LIN {X -15.690,Y -24.253,Z -48.585,A -90.000,B 90.000,C 0.000} C_DIS
LIN {X -14.979,Y -24.271,Z -48.414,A -90.000,B 90.000,C 0.000} C_DIS
LIN {X -14.534,Y -24.273,Z -48.316,A -90.000,B 90.000,C 0.000} C_DIS
LIN {X -13.675,Y -24.281,Z -48.156,A -90.000,B 90.000,C 0.000} C_DIS
LIN {X -13.403,Y -24.283,Z -48.108,A -90.000,B 90.000,C 0.000} C_DIS
LIN {X -13.192,Y -24.287,Z -48.076,A -90.000,B 90.000,C 0.000} C_DIS
LIN {X -13.001,Y -24.291,Z -48.054,A -90.000,B 90.000,C 0.000} C_DIS
LIN {X -12.088,Y -24.285,Z -47.948,A -90.000,B 90.000,C 0.000} C_DIS
LIN {X -11.996,Y -24.284,Z -47.939,A -90.000,B 90.000,C 0.000} C_DIS
LIN {X -10.985,Y -24.286,Z -47.870,A -90.000,B 90.000,C 0.000} C_DIS
LIN {X -10.430,Y -24.283,Z -47.833,A -90.000,B 90.000,C 0.000} C_DIS
LIN {X -10.008,Y -24.276,Z -47.814,A -90.000,B 90.000,C 0.000} C_DIS
LIN {X -9.074,Y -24.265,Z -47.794,A -90.000,B 90.000,C 0.000} C_DIS
LIN {X -8.874,Y -24.263,Z -47.795,A -90.000,B 90.000,C 0.000} C_DIS
LIN {X -8.324,Y -24.259,Z -47.794,A -90.000,B 90.000,C 0.000} C_DIS
LIN {X -8.099,Y -24.253,Z -47.798,A -90.000,B 90.000,C 0.000} C_DIS
LIN {X -6.871,Y -24.218,Z -47.835,A -90.000,B 90.000,C 0.000} C_DIS
LIN {X -5.951,Y -24.176,Z -47.868,A -90.000,B 90.000,C 0.000} C_DIS
LIN {X -5.359,Y -24.150,Z -47.900,A -90.000,B 90.000,C 0.000} C_DIS
LIN {X -3.919,Y -24.078,Z -48.003,A -90.000,B 90.000,C 0.000} C_DIS
LIN {X -3.281,Y -24.035,Z -48.050,A -90.000,B 90.000,C 0.000} C_DIS
LIN {X -3.006,Y -24.019,Z -48.078,A -90.000,B 90.000,C 0.000} C_DIS
LIN {X -2.826,Y -24.007,Z -48.091,A -90.000,B 90.000,C 0.000} C_DIS
LIN {X -2.559,Y -23.983,Z -48.112,A -90.000,B 90.000,C 0.000} C_DIS
LIN {X -1.553,Y -23.901,Z -48.211,A -90.000,B 90.000,C 0.000} C_DIS
LIN {X -0.357,Y -23.796,Z -48.335,A -90.000,B 90.000,C 0.000} C_DIS
LIN {X -0.072,Y -23.770,Z -48.373,A -90.000,B 90.000,C 0.000} C_DIS
LIN {X 0.616,Y -23.686,Z -48.423,A -90.000,B 90.000,C 0.000} C_DIS
LIN {X 0.820,Y -23.658,Z -48.442,A -90.000,B 90.000,C 0.000} C_DIS
LIN {X 1.112,Y -23.624,Z -48.468,A -90.000,B 90.000,C 0.000} C_DIS
LIN {X 1.553,Y -23.560,Z -48.482,A -90.000,B 90.000,C 0.000} C_DIS
LIN {X 2.189,Y -23.460,Z -48.509,A -90.000,B 90.000,C 0.000} C_DIS
LIN {X 2.579,Y -23.392,Z -48.514,A -90.000,B 90.000,C 0.000} C_DIS
LIN {X 3.096,Y -23.308,Z -48.519,A -90.000,B 90.000,C 0.000} C_DIS
LIN {X 3.096,Y -60.000,Z -48.519,A -90.000,B 90.000,C 0.000} C_DIS
LIN {X -32.585,Y -60.000,Z -45.788,A -90.000,B 90.000,C 0.000} C_DIS
LIN {X -32.585,Y -23.308,Z -45.788,A -90.000,B 90.000,C 0.000} C_DIS
LIN {X -32.505,Y -23.313,Z -45.784,A -90.000,B 90.000,C 0.000} C_DIS
LIN {X -31.998,Y -23.345,Z -45.829,A -90.000,B 90.000,C 0.000} C_DIS
LIN {X -31.484,Y -23.377,Z -45.944,A -90.000,B 90.000,C 0.000} C_DIS
LIN {X -30.921,Y -23.413,Z -46.084,A -90.000,B 90.000,C 0.000} C_DIS
LIN {X -30.620,Y -23.432,Z -46.161,A -90.000,B 90.000,C 0.000} C_DIS
LIN {X -29.471,Y -23.490,Z -46.457,A -90.000,B 90.000,C 0.000} C_DIS
LIN {X -28.623,Y -23.534,Z -46.679,A -90.000,B 90.000,C 0.000} C_DIS
LIN {X -27.966,Y -23.569,Z -46.858,A -90.000,B 90.000,C 0.000} C_DIS
LIN {X -27.371,Y -23.600,Z -47.027,A -90.000,B 90.000,C 0.000} C_DIS
LIN {X -26.595,Y -23.630,Z -47.249,A -90.000,B 90.000,C 0.000} C_DIS
LIN {X -25.870,Y -23.674,Z -47.454,A -90.000,B 90.000,C 0.000} C_DIS
LIN {X -24.845,Y -23.735,Z -47.733,A -90.000,B 90.000,C 0.000} C_DIS
LIN {X -24.579,Y -23.747,Z -47.807,A -90.000,B 90.000,C 0.000} C_DIS
LIN {X -23.879,Y -23.794,Z -48.000,A -90.000,B 90.000,C 0.000} C_DIS
LIN {X -23.725,Y -23.804,Z -48.041,A -90.000,B 90.000,C 0.000} C_DIS
LIN {X -22.667,Y -23.874,Z -48.311,A -90.000,B 90.000,C 0.000} C_DIS
LIN {X -22.222,Y -23.905,Z -48.432,A -90.000,B 90.000,C 0.000} C_DIS
LIN {X -21.863,Y -23.929,Z -48.510,A -90.000,B 90.000,C 0.000} C_DIS
LIN {X -21.455,Y -23.955,Z -48.592,A -90.000,B 90.000,C 0.000} C_DIS
LIN {X -21.255,Y -23.968,Z -48.635,A -90.000,B 90.000,C 0.000} C_DIS
LIN {X -21.041,Y -23.972,Z -48.532,A -90.000,B 90.000,C 0.000} C_DIS
LIN {X -20.633,Y -23.979,Z -48.352,A -90.000,B 90.000,C 0.000} C_DIS
LIN {X -20.360,Y -23.979,Z -48.218,A -90.000,B 90.000,C 0.000} C_DIS
LIN {X -19.794,Y -23.981,Z -47.962,A -90.000,B 90.000,C 0.000} C_DIS
LIN {X -19.288,Y -23.984,Z -47.740,A -90.000,B 90.000,C 0.000} C_DIS
LIN {X -18.693,Y -23.989,Z -47.495,A -90.000,B 90.000,C 0.000} C_DIS
LIN {X -18.571,Y -23.990,Z -47.448,A -90.000,B 90.000,C 0.000} C_DIS
LIN {X -18.128,Y -23.997,Z -47.278,A -90.000,B 90.000,C 0.000} C_DIS
LIN {X -17.827,Y -23.998,Z -47.165,A -90.000,B 90.000,C 0.000} C_DIS
LIN {X -17.635,Y -23.992,Z -47.095,A -90.000,B 90.000,C 0.000} C_DIS
LIN {X -17.171,Y -23.976,Z -46.936,A -90.000,B 90.000,C 0.000} C_DIS
LIN {X -16.972,Y -23.970,Z -46.873,A -90.000,B 90.000,C 0.000} C_DIS
LIN {X -16.791,Y -23.966,Z -46.823,A -90.000,B 90.000,C 0.000} C_DIS
LIN {X -16.610,Y -23.962,Z -46.776,A -90.000,B 90.000,C 0.000} C_DIS
LIN {X -16.390,Y -23.958,Z -46.723,A -90.000,B 90.000,C 0.000} C_DIS
LIN {X -16.098,Y -23.953,Z -46.650,A -90.000,B 90.000,C 0.000} C_DIS
LIN {X -15.459,Y -23.940,Z -46.501,A -90.000,B 90.000,C 0.000} C_DIS
LIN {X -14.891,Y -23.930,Z -46.378,A -90.000,B 90.000,C 0.000} C_DIS
LIN {X -14.327,Y -23.923,Z -46.276,A -90.000,B 90.000,C 0.000} C_DIS
LIN {X -14.012,Y -23.915,Z -46.219,A -90.000,B 90.000,C 0.000} C_DIS
LIN {X -13.695,Y -23.908,Z -46.166,A -90.000,B 90.000,C 0.000} C_DIS
LIN {X -13.405,Y -23.902,Z -46.125,A -90.000,B 90.000,C 0.000} C_DIS
LIN {X -12.856,Y -23.894,Z -46.063,A -90.000,B 90.000,C 0.000} C_DIS
LIN {X -12.269,Y -23.874,Z -45.999,A -90.000,B 90.000,C 0.000} C_DIS
LIN {X -12.130,Y -23.869,Z -45.988,A -90.000,B 90.000,C 0.000} C_DIS
LIN {X -11.523,Y -23.849,Z -45.950,A -90.000,B 90.000,C 0.000} C_DIS
LIN {X -10.523,Y -23.813,Z -45.891,A -90.000,B 90.000,C 0.000} C_DIS
LIN {X -10.335,Y -23.807,Z -45.884,A -90.000,B 90.000,C 0.000} C_DIS
LIN {X -10.056,Y -23.794,Z -45.874,A -90.000,B 90.000,C 0.000} C_DIS
LIN {X -9.071,Y -23.756,Z -45.860,A -90.000,B 90.000,C 0.000} C_DIS
LIN {X -8.242,Y -23.727,Z -45.867,A -90.000,B 90.000,C 0.000} C_DIS
LIN {X -7.898,Y -23.712,Z -45.877,A -90.000,B 90.000,C 0.000} C_DIS
LIN {X -6.829,Y -23.656,Z -45.916,A -90.000,B 90.000,C 0.000} C_DIS
LIN {X -5.872,Y -23.593,Z -45.956,A -90.000,B 90.000,C 0.000} C_DIS
LIN {X -5.253,Y -23.547,Z -45.996,A -90.000,B 90.000,C 0.000} C_DIS
LIN {X -4.815,Y -23.517,Z -46.030,A -90.000,B 90.000,C 0.000} C_DIS
LIN {X -3.187,Y -23.355,Z -46.172,A -90.000,B 90.000,C 0.000} C_DIS
LIN {X -2.890,Y -23.324,Z -46.206,A -90.000,B 90.000,C 0.000} C_DIS
LIN {X -2.747,Y -23.308,Z -46.218,A -90.000,B 90.000,C 0.000} C_DIS
LIN {X -2.747,Y -60.000,Z -46.218,A -90.000,B 90.000,C 0.000} C_DIS
LIN {X -28.775,Y -60.000,Z -44.581,A -90.000,B 90.000,C 0.000} C_DIS
LIN {X -28.775,Y -23.308,Z -44.581,A -90.000,B 90.000,C 0.000} C_DIS
LIN {X -27.940,Y -23.354,Z -44.801,A -90.000,B 90.000,C 0.000} C_DIS
LIN {X -27.677,Y -23.366,Z -44.873,A -90.000,B 90.000,C 0.000} C_DIS
LIN {X -27.412,Y -23.377,Z -44.946,A -90.000,B 90.000,C 0.000} C_DIS
LIN {X -26.438,Y -23.416,Z -45.224,A -90.000,B 90.000,C 0.000} C_DIS
LIN {X -25.243,Y -23.500,Z -45.560,A -90.000,B 90.000,C 0.000} C_DIS
LIN {X -24.377,Y -23.540,Z -45.797,A -90.000,B 90.000,C 0.000} C_DIS
LIN {X -23.210,Y -23.631,Z -46.116,A -90.000,B 90.000,C 0.000} C_DIS
LIN {X -22.965,Y -23.648,Z -46.179,A -90.000,B 90.000,C 0.000} C_DIS
LIN {X -22.513,Y -23.673,Z -46.294,A -90.000,B 90.000,C 0.000} C_DIS
LIN {X -22.132,Y -23.703,Z -46.391,A -90.000,B 90.000,C 0.000} C_DIS
LIN {X -21.755,Y -23.733,Z -46.495,A -90.000,B 90.000,C 0.000} C_DIS
LIN {X -21.480,Y -23.754,Z -46.554,A -90.000,B 90.000,C 0.000} C_DIS
LIN {X -21.262,Y -23.752,Z -46.447,A -90.000,B 90.000,C 0.000} C_DIS
LIN {X -21.012,Y -23.750,Z -46.332,A -90.000,B 90.000,C 0.000} C_DIS
LIN {X -20.884,Y -23.746,Z -46.275,A -90.000,B 90.000,C 0.000} C_DIS
LIN {X -20.466,Y -23.723,Z -46.091,A -90.000,B 90.000,C 0.000} C_DIS
LIN {X -20.040,Y -23.701,Z -45.909,A -90.000,B 90.000,C 0.000} C_DIS
LIN {X -19.444,Y -23.672,Z -45.669,A -90.000,B 90.000,C 0.000} C_DIS
LIN {X -18.658,Y -23.639,Z -45.376,A -90.000,B 90.000,C 0.000} C_DIS
LIN {X -18.327,Y -23.625,Z -45.254,A -90.000,B 90.000,C 0.000} C_DIS
LIN {X -17.772,Y -23.605,Z -45.064,A -90.000,B 90.000,C 0.000} C_DIS
LIN {X -17.669,Y -23.602,Z -45.032,A -90.000,B 90.000,C 0.000} C_DIS
LIN {X -17.499,Y -23.597,Z -44.980,A -90.000,B 90.000,C 0.000} C_DIS
LIN {X -17.320,Y -23.592,Z -44.931,A -90.000,B 90.000,C 0.000} C_DIS
LIN {X -16.958,Y -23.568,Z -44.842,A -90.000,B 90.000,C 0.000} C_DIS
LIN {X -16.506,Y -23.540,Z -44.735,A -90.000,B 90.000,C 0.000} C_DIS
LIN {X -15.878,Y -23.503,Z -44.595,A -90.000,B 90.000,C 0.000} C_DIS
LIN {X -15.310,Y -23.472,Z -44.477,A -90.000,B 90.000,C 0.000} C_DIS
LIN {X -14.339,Y -23.429,Z -44.307,A -90.000,B 90.000,C 0.000} C_DIS
LIN {X -13.945,Y -23.412,Z -44.244,A -90.000,B 90.000,C 0.000} C_DIS
LIN {X -13.628,Y -23.395,Z -44.203,A -90.000,B 90.000,C 0.000} C_DIS
LIN {X -12.619,Y -23.342,Z -44.099,A -90.000,B 90.000,C 0.000} C_DIS
LIN {X -12.445,Y -23.328,Z -44.083,A -90.000,B 90.000,C 0.000} C_DIS
LIN {X -12.266,Y -23.316,Z -44.070,A -90.000,B 90.000,C 0.000} C_DIS
LIN {X -12.141,Y -23.308,Z -44.064,A -90.000,B 90.000,C 0.000} C_DIS
LIN {X -12.141,Y -60.000,Z -44.064,A -90.000,B 90.000,C 0.000} C_DIS
LIN {X -22.320,Y -60.000,Z -44.311,A -90.000,B 90.000,C 0.000} C_DIS
LIN {X -22.320,Y -23.308,Z -44.311,A -90.000,B 90.000,C 0.000} C_DIS
LIN {X -22.204,Y -23.316,Z -44.340,A -90.000,B 90.000,C 0.000} C_DIS
LIN {X -21.668,Y -23.364,Z -44.475,A -90.000,B 90.000,C 0.000} C_DIS
LIN {X -21.152,Y -23.332,Z -44.250,A -90.000,B 90.000,C 0.000} C_DIS
LIN {X -20.759,Y -23.308,Z -44.084,A -90.000,B 90.000,C 0.000} C_DIS
LIN {X -20.759,Y -60.000,Z -44.084,A -90.000,B 90.000,C 0.000} C_DIS
LIN {X -95.711,Y -60.000,Z -40.754,A -90.000,B 90.000,C 0.000} C_DIS
LIN {X -95.711,Y -23.308,Z -40.754,A -90.000,B 90.000,C 0.000} C_DIS
LIN {X -95.404,Y -23.376,Z -40.730,A -90.000,B 90.000,C 0.000} C_DIS
LIN {X -95.125,Y -23.439,Z -40.718,A -90.000,B 90.000,C 0.000} C_DIS
LIN {X -94.697,Y -23.539,Z -40.707,A -90.000,B 90.000,C 0.000} C_DIS
LIN {X -94.412,Y -23.607,Z -40.709,A -90.000,B 90.000,C 0.000} C_DIS
LIN {X -94.097,Y -23.689,Z -40.720,A -90.000,B 90.000,C 0.000} C_DIS
LIN {X -93.821,Y -23.753,Z -40.682,A -90.000,B 90.000,C 0.000} C_DIS
LIN {X -93.679,Y -23.787,Z -40.667,A -90.000,B 90.000,C 0.000} C_DIS
LIN {X -93.582,Y -23.810,Z -40.659,A -90.000,B 90.000,C 0.000} C_DIS
LIN {X -93.062,Y -23.940,Z -40.640,A -90.000,B 90.000,C 0.000} C_DIS
LIN {X -92.947,Y -23.969,Z -40.636,A -90.000,B 90.000,C 0.000} C_DIS
LIN {X -92.686,Y -24.037,Z -40.636,A -90.000,B 90.000,C 0.000} C_DIS
LIN {X -92.525,Y -24.079,Z -40.642,A -90.000,B 90.000,C 0.000} C_DIS
LIN {X -92.268,Y -24.147,Z -40.654,A -90.000,B 90.000,C 0.000} C_DIS
LIN {X -91.922,Y -24.239,Z -40.676,A -90.000,B 90.000,C 0.000} C_DIS
LIN {X -91.828,Y -24.217,Z -40.402,A -90.000,B 90.000,C 0.000} C_DIS
LIN {X -91.794,Y -24.207,Z -40.309,A -90.000,B 90.000,C 0.000} C_DIS
LIN {X -91.725,Y -24.191,Z -40.113,A -90.000,B 90.000,C 0.000} C_DIS
LIN {X -91.669,Y -24.181,Z -39.970,A -90.000,B 90.000,C 0.000} C_DIS
LIN {X -91.619,Y -24.175,Z -39.854,A -90.000,B 90.000,C 0.000} C_DIS
LIN {X -91.566,Y -24.169,Z -39.741,A -90.000,B 90.000,C 0.000} C_DIS
LIN {X -91.504,Y -24.165,Z -39.621,A -90.000,B 90.000,C 0.000} C_DIS
LIN {X -91.441,Y -24.153,Z -39.505,A -90.000,B 90.000,C 0.000} C_DIS
LIN {X -91.356,Y -24.139,Z -39.362,A -90.000,B 90.000,C 0.000} C_DIS
LIN {X -91.326,Y -24.131,Z -39.314,A -90.000,B 90.000,C 0.000} C_DIS
LIN {X -91.245,Y -24.118,Z -39.180,A -90.000,B 90.000,C 0.000} C_DIS
LIN {X -91.203,Y -24.112,Z -39.116,A -90.000,B 90.000,C 0.000} C_DIS
LIN {X -91.034,Y -24.087,Z -38.886,A -90.000,B 90.000,C 0.000} C_DIS
LIN {X -90.958,Y -24.072,Z -38.743,A -90.000,B 90.000,C 0.000} C_DIS
LIN {X -90.838,Y -24.039,Z -38.550,A -90.000,B 90.000,C 0.000} C_DIS
LIN {X -90.746,Y -24.015,Z -38.415,A -90.000,B 90.000,C 0.000} C_DIS
LIN {X -90.547,Y -23.961,Z -38.143,A -90.000,B 90.000,C 0.000} C_DIS
LIN {X -90.460,Y -23.947,Z -38.029,A -90.000,B 90.000,C 0.000} C_DIS
LIN {X -90.374,Y -23.936,Z -37.924,A -90.000,B 90.000,C 0.000} C_DIS
LIN {X -90.278,Y -23.926,Z -37.813,A -90.000,B 90.000,C 0.000} C_DIS
LIN {X -90.089,Y -23.895,Z -37.621,A -90.000,B 90.000,C 0.000} C_DIS
LIN {X -89.954,Y -23.869,Z -37.492,A -90.000,B 90.000,C 0.000} C_DIS
LIN {X -89.904,Y -23.863,Z -37.443,A -90.000,B 90.000,C 0.000} C_DIS
LIN {X -89.803,Y -23.853,Z -37.352,A -90.000,B 90.000,C 0.000} C_DIS
LIN {X -89.654,Y -23.839,Z -37.224,A -90.000,B 90.000,C 0.000} C_DIS
LIN {X -89.505,Y -23.828,Z -37.109,A -90.000,B 90.000,C 0.000} C_DIS
LIN {X -89.400,Y -23.817,Z -37.035,A -90.000,B 90.000,C 0.000} C_DIS
LIN {X -89.138,Y -23.799,Z -36.847,A -90.000,B 90.000,C 0.000} C_DIS
LIN {X -89.084,Y -23.790,Z -36.797,A -90.000,B 90.000,C 0.000} C_DIS
LIN {X -88.968,Y -23.771,Z -36.698,A -90.000,B 90.000,C 0.000} C_DIS
LIN {X -88.747,Y -23.744,Z -36.523,A -90.000,B 90.000,C 0.000} C_DIS
LIN {X -88.371,Y -23.709,Z -36.261,A -90.000,B 90.000,C 0.000} C_DIS
LIN {X -88.226,Y -23.699,Z -36.167,A -90.000,B 90.000,C 0.000} C_DIS
LIN {X -88.132,Y -23.696,Z -36.112,A -90.000,B 90.000,C 0.000} C_DIS
LIN {X -87.910,Y -23.694,Z -35.987,A -90.000,B 90.000,C 0.000} C_DIS
LIN {X -87.694,Y -23.697,Z -35.875,A -90.000,B 90.000,C 0.000} C_DIS
LIN {X -87.253,Y -23.682,Z -35.604,A -90.000,B 90.000,C 0.000} C_DIS
LIN {X -87.176,Y -23.680,Z -35.559,A -90.000,B 90.000,C 0.000} C_DIS
LIN {X -86.953,Y -23.677,Z -35.437,A -90.000,B 90.000,C 0.000} C_DIS
LIN {X -86.816,Y -23.677,Z -35.368,A -90.000,B 90.000,C 0.000} C_DIS
LIN {X -86.698,Y -23.684,Z -35.304,A -90.000,B 90.000,C 0.000} C_DIS
LIN {X -86.576,Y -23.704,Z -35.237,A -90.000,B 90.000,C 0.000} C_DIS
LIN {X -86.405,Y -23.727,Z -35.152,A -90.000,B 90.000,C 0.000} C_DIS
LIN {X -86.301,Y -23.742,Z -35.107,A -90.000,B 90.000,C 0.000} C_DIS
LIN {X -86.104,Y -23.770,Z -35.028,A -90.000,B 90.000,C 0.000} C_DIS
LIN {X -85.996,Y -23.785,Z -34.990,A -90.000,B 90.000,C 0.000} C_DIS
LIN {X -85.717,Y -23.820,Z -34.894,A -90.000,B 90.000,C 0.000} C_DIS
LIN {X -85.064,Y -23.902,Z -34.688,A -90.000,B 90.000,C 0.000} C_DIS
LIN {X -84.998,Y -23.910,Z -34.665,A -90.000,B 90.000,C 0.000} C_DIS
LIN {X -84.512,Y -23.958,Z -34.499,A -90.000,B 90.000,C 0.000} C_DIS
LIN {X -84.366,Y -23.973,Z -34.452,A -90.000,B 90.000,C 0.000} C_DIS
LIN {X -84.135,Y -23.992,Z -34.378,A -90.000,B 90.000,C 0.000} C_DIS
LIN {X -84.049,Y -24.002,Z -34.353,A -90.000,B 90.000,C 0.000} C_DIS
LIN {X -83.904,Y -24.017,Z -34.314,A -90.000,B 90.000,C 0.000} C_DIS
LIN {X -83.669,Y -24.044,Z -34.261,A -90.000,B 90.000,C 0.000} C_DIS
LIN {X -83.463,Y -24.068,Z -34.227,A -90.000,B 90.000,C 0.000} C_DIS
LIN {X -83.165,Y -24.104,Z -34.187,A -90.000,B 90.000,C 0.000} C_DIS
LIN {X -83.013,Y -24.122,Z -34.173,A -90.000,B 90.000,C 0.000} C_DIS
LIN {X -82.811,Y -24.142,Z -34.160,A -90.000,B 90.000,C 0.000} C_DIS
LIN {X -81.766,Y -24.254,Z -34.100,A -90.000,B 90.000,C 0.000} C_DIS
LIN {X -81.587,Y -24.268,Z -34.092,A -90.000,B 90.000,C 0.000} C_DIS
LIN {X -81.311,Y -24.285,Z -34.078,A -90.000,B 90.000,C 0.000} C_DIS
LIN {X -81.094,Y -24.301,Z -34.074,A -90.000,B 90.000,C 0.000} C_DIS
LIN {X -80.876,Y -24.317,Z -34.077,A -90.000,B 90.000,C 0.000} C_DIS
LIN {X -80.753,Y -24.325,Z -34.081,A -90.000,B 90.000,C 0.000} C_DIS
LIN {X -80.316,Y -24.356,Z -34.112,A -90.000,B 90.000,C 0.000} C_DIS
LIN {X -80.028,Y -24.375,Z -34.145,A -90.000,B 90.000,C 0.000} C_DIS
LIN {X -79.790,Y -24.379,Z -34.178,A -90.000,B 90.000,C 0.000} C_DIS
LIN {X -79.303,Y -24.376,Z -34.251,A -90.000,B 90.000,C 0.000} C_DIS
LIN {X -78.837,Y -24.372,Z -34.323,A -90.000,B 90.000,C 0.000} C_DIS
LIN {X -78.575,Y -24.369,Z -34.362,A -90.000,B 90.000,C 0.000} C_DIS
LIN {X -78.371,Y -24.366,Z -34.396,A -90.000,B 90.000,C 0.000} C_DIS
LIN {X -78.171,Y -24.360,Z -34.436,A -90.000,B 90.000,C 0.000} C_DIS
LIN {X -77.664,Y -24.319,Z -34.565,A -90.000,B 90.000,C 0.000} C_DIS
LIN {X -77.527,Y -24.308,Z -34.603,A -90.000,B 90.000,C 0.000} C_DIS
LIN {X -76.621,Y -24.210,Z -34.862,A -90.000,B 90.000,C 0.000} C_DIS
LIN {X -76.352,Y -24.182,Z -34.940,A -90.000,B 90.000,C 0.000} C_DIS
LIN {X -76.038,Y -24.153,Z -35.031,A -90.000,B 90.000,C 0.000} C_DIS
LIN {X -75.954,Y -24.146,Z -35.059,A -90.000,B 90.000,C 0.000} C_DIS
LIN {X -75.336,Y -24.059,Z -35.270,A -90.000,B 90.000,C 0.000} C_DIS
LIN {X -75.055,Y -24.015,Z -35.369,A -90.000,B 90.000,C 0.000} C_DIS
LIN {X -74.477,Y -23.967,Z -35.562,A -90.000,B 90.000,C 0.000} C_DIS
LIN {X -73.802,Y -23.909,Z -35.764,A -90.000,B 90.000,C 0.000} C_DIS
LIN {X -73.585,Y -23.884,Z -35.832,A -90.000,B 90.000,C 0.000} C_DIS
LIN {X -72.583,Y -23.813,Z -36.131,A -90.000,B 90.000,C 0.000} C_DIS
LIN {X -72.099,Y -23.794,Z -36.270,A -90.000,B 90.000,C 0.000} C_DIS
LIN {X -71.852,Y -23.780,Z -36.342,A -90.000,B 90.000,C 0.000} C_DIS
LIN {X -71.586,Y -23.758,Z -36.423,A -90.000,B 90.000,C 0.000} C_DIS
LIN {X -71.224,Y -23.733,Z -36.546,A -90.000,B 90.000,C 0.000} C_DIS
LIN {X -69.912,Y -23.680,Z -36.977,A -90.000,B 90.000,C 0.000} C_DIS
LIN {X -69.703,Y -23.674,Z -37.053,A -90.000,B 90.000,C 0.000} C_DIS
LIN {X -67.916,Y -23.609,Z -37.754,A -90.000,B 90.000,C 0.000} C_DIS
LIN {X -67.475,Y -23.601,Z -37.944,A -90.000,B 90.000,C 0.000} C_DIS
LIN {X -67.275,Y -23.600,Z -38.034,A -90.000,B 90.000,C 0.000} C_DIS
LIN {X -66.096,Y -23.581,Z -38.568,A -90.000,B 90.000,C 0.000} C_DIS
LIN {X -65.374,Y -23.570,Z -38.895,A -90.000,B 90.000,C 0.000} C_DIS
LIN {X -65.123,Y -23.567,Z -39.012,A -90.000,B 90.000,C 0.000} C_DIS
LIN {X -64.632,Y -23.569,Z -39.237,A -90.000,B 90.000,C 0.000} C_DIS
LIN {X -63.049,Y -23.568,Z -39.976,A -90.000,B 90.000,C 0.000} C_DIS
LIN {X -62.587,Y -23.563,Z -40.182,A -90.000,B 90.000,C 0.000} C_DIS
LIN {X -61.622,Y -23.570,Z -40.601,A -90.000,B 90.000,C 0.000} C_DIS
LIN {X -60.883,Y -23.573,Z -40.925,A -90.000,B 90.000,C 0.000} C_DIS
LIN {X -59.965,Y -23.555,Z -41.283,A -90.000,B 90.000,C 0.000} C_DIS
LIN {X -58.440,Y -23.556,Z -41.863,A -90.000,B 90.000,C 0.000} C_DIS
LIN {X -57.686,Y -23.533,Z -42.100,A -90.000,B 90.000,C 0.000} C_DIS
LIN {X -57.271,Y -23.524,Z -42.228,A -90.000,B 90.000,C 0.000} C_DIS
LIN {X -56.299,Y -23.512,Z -42.523,A -90.000,B 90.000,C 0.000} C_DIS
LIN {X -55.979,Y -23.509,Z -42.624,A -90.000,B 90.000,C 0.000} C_DIS
LIN {X -54.824,Y -23.462,Z -42.911,A -90.000,B 90.000,C 0.000} C_DIS
LIN {X -54.566,Y -23.454,Z -42.978,A -90.000,B 90.000,C 0.000} C_DIS
LIN {X -53.632,Y -23.437,Z -43.217,A -90.000,B 90.000,C 0.000} C_DIS
LIN {X -53.189,Y -23.414,Z -43.304,A -90.000,B 90.000,C 0.000} C_DIS
LIN {X -52.188,Y -23.372,Z -43.522,A -90.000,B 90.000,C 0.000} C_DIS
LIN {X -51.677,Y -23.361,Z -43.648,A -90.000,B 90.000,C 0.000} C_DIS
LIN {X -50.718,Y -23.347,Z -43.882,A -90.000,B 90.000,C 0.000} C_DIS
LIN {X -50.007,Y -23.330,Z -44.041,A -90.000,B 90.000,C 0.000} C_DIS
LIN {X -49.018,Y -23.308,Z -44.257,A -90.000,B 90.000,C 0.000} C_DIS
LIN {X -49.018,Y -60.000,Z -44.257,A -90.000,B 90.000,C 0.000} C_DIS
LIN {X -88.889,Y -60.000,Z -34.286,A -90.000,B 90.000,C 0.000} C_DIS
LIN {X -88.889,Y -23.308,Z -34.286,A -90.000,B 90.000,C 0.000} C_DIS
LIN {X -88.778,Y -23.327,Z -34.222,A -90.000,B 90.000,C 0.000} C_DIS
LIN {X -88.666,Y -23.346,Z -34.161,A -90.000,B 90.000,C 0.000} C_DIS
LIN {X -88.534,Y -23.367,Z -34.075,A -90.000,B 90.000,C 0.000} C_DIS
LIN {X -88.241,Y -23.405,Z -33.888,A -90.000,B 90.000,C 0.000} C_DIS
LIN {X -88.132,Y -23.419,Z -33.822,A -90.000,B 90.000,C 0.000} C_DIS
LIN {X -87.851,Y -23.453,Z -33.664,A -90.000,B 90.000,C 0.000} C_DIS
LIN {X -87.674,Y -23.475,Z -33.571,A -90.000,B 90.000,C 0.000} C_DIS
LIN {X -87.558,Y -23.485,Z -33.508,A -90.000,B 90.000,C 0.000} C_DIS
LIN {X -87.382,Y -23.494,Z -33.417,A -90.000,B 90.000,C 0.000} C_DIS
LIN {X -87.268,Y -23.500,Z -33.362,A -90.000,B 90.000,C 0.000} C_DIS
LIN {X -87.116,Y -23.508,Z -33.294,A -90.000,B 90.000,C 0.000} C_DIS
LIN {X -86.979,Y -23.516,Z -33.238,A -90.000,B 90.000,C 0.000} C_DIS
LIN {X -86.761,Y -23.529,Z -33.155,A -90.000,B 90.000,C 0.000} C_DIS
LIN {X -86.511,Y -23.545,Z -33.069,A -90.000,B 90.000,C 0.000} C_DIS
LIN {X -86.235,Y -23.568,Z -32.978,A -90.000,B 90.000,C 0.000} C_DIS
LIN {X -85.622,Y -23.609,Z -32.788,A -90.000,B 90.000,C 0.000} C_DIS
LIN {X -85.221,Y -23.633,Z -32.655,A -90.000,B 90.000,C 0.000} C_DIS
LIN {X -84.885,Y -23.675,Z -32.542,A -90.000,B 90.000,C 0.000} C_DIS
LIN {X -84.715,Y -23.696,Z -32.487,A -90.000,B 90.000,C 0.000} C_DIS
LIN {X -84.589,Y -23.712,Z -32.449,A -90.000,B 90.000,C 0.000} C_DIS
LIN {X -84.319,Y -23.747,Z -32.376,A -90.000,B 90.000,C 0.000} C_DIS
LIN {X -84.073,Y -23.788,Z -32.319,A -90.000,B 90.000,C 0.000} C_DIS
LIN {X -83.965,Y -23.806,Z -32.298,A -90.000,B 90.000,C 0.000} C_DIS
LIN {X -83.702,Y -23.850,Z -32.253,A -90.000,B 90.000,C 0.000} C_DIS
LIN {X -83.406,Y -23.900,Z -32.212,A -90.000,B 90.000,C 0.000} C_DIS
LIN {X -83.176,Y -23.940,Z -32.188,A -90.000,B 90.000,C 0.000} C_DIS
LIN {X -82.798,Y -24.007,Z -32.161,A -90.000,B 90.000,C 0.000} C_DIS
LIN {X -82.322,Y -24.090,Z -32.132,A -90.000,B 90.000,C 0.000} C_DIS
LIN {X -81.879,Y -24.162,Z -32.105,A -90.000,B 90.000,C 0.000} C_DIS
LIN {X -81.618,Y -24.203,Z -32.092,A -90.000,B 90.000,C 0.000} C_DIS
LIN {X -81.411,Y -24.229,Z -32.082,A -90.000,B 90.000,C 0.000} C_DIS
LIN {X -81.065,Y -24.268,Z -32.074,A -90.000,B 90.000,C 0.000} C_DIS
LIN {X -80.767,Y -24.303,Z -32.079,A -90.000,B 90.000,C 0.000} C_DIS
LIN {X -80.612,Y -24.323,Z -32.086,A -90.000,B 90.000,C 0.000} C_DIS
LIN {X -80.222,Y -24.371,Z -32.114,A -90.000,B 90.000,C 0.000} C_DIS
LIN {X -80.090,Y -24.383,Z -32.125,A -90.000,B 90.000,C 0.000} C_DIS
LIN {X -79.758,Y -24.412,Z -32.164,A -90.000,B 90.000,C 0.000} C_DIS
LIN {X -79.546,Y -24.429,Z -32.193,A -90.000,B 90.000,C 0.000} C_DIS
LIN {X -79.200,Y -24.444,Z -32.245,A -90.000,B 90.000,C 0.000} C_DIS
LIN {X -79.004,Y -24.448,Z -32.275,A -90.000,B 90.000,C 0.000} C_DIS
LIN {X -78.188,Y -24.442,Z -32.400,A -90.000,B 90.000,C 0.000} C_DIS
LIN {X -78.032,Y -24.438,Z -32.426,A -90.000,B 90.000,C 0.000} C_DIS
LIN {X -77.969,Y -24.434,Z -32.438,A -90.000,B 90.000,C 0.000} C_DIS
LIN {X -77.785,Y -24.419,Z -32.474,A -90.000,B 90.000,C 0.000} C_DIS
LIN {X -77.638,Y -24.407,Z -32.508,A -90.000,B 90.000,C 0.000} C_DIS
LIN {X -77.098,Y -24.355,Z -32.647,A -90.000,B 90.000,C 0.000} C_DIS
LIN {X -76.573,Y -24.302,Z -32.796,A -90.000,B 90.000,C 0.000} C_DIS
LIN {X -76.436,Y -24.283,Z -32.835,A -90.000,B 90.000,C 0.000} C_DIS
LIN {X -76.069,Y -24.222,Z -32.940,A -90.000,B 90.000,C 0.000} C_DIS
LIN {X -75.819,Y -24.176,Z -33.012,A -90.000,B 90.000,C 0.000} C_DIS
LIN {X -75.618,Y -24.137,Z -33.071,A -90.000,B 90.000,C 0.000} C_DIS
LIN {X -75.424,Y -24.099,Z -33.129,A -90.000,B 90.000,C 0.000} C_DIS
LIN {X -75.182,Y -24.043,Z -33.211,A -90.000,B 90.000,C 0.000} C_DIS
LIN {X -74.616,Y -23.897,Z -33.409,A -90.000,B 90.000,C 0.000} C_DIS
LIN {X -73.871,Y -23.698,Z -33.674,A -90.000,B 90.000,C 0.000} C_DIS
LIN {X -73.225,Y -23.527,Z -33.888,A -90.000,B 90.000,C 0.000} C_DIS
LIN {X -73.049,Y -23.476,Z -33.949,A -90.000,B 90.000,C 0.000} C_DIS
LIN {X -72.827,Y -23.429,Z -34.022,A -90.000,B 90.000,C 0.000} C_DIS
LIN {X -72.333,Y -23.308,Z -34.192,A -90.000,B 90.000,C 0.000} C_DIS
LIN {X -72.333,Y -60.000,Z -34.192,A -90.000,B 90.000,C 0.000} C_DIS
LIN {X -85.759,Y -60.000,Z -30.755,A -90.000,B 90.000,C 0.000} C_DIS
LIN {X -85.759,Y -23.308,Z -30.755,A -90.000,B 90.000,C 0.000} C_DIS
LIN {X -85.664,Y -23.324,Z -30.723,A -90.000,B 90.000,C 0.000} C_DIS
LIN {X -85.255,Y -23.408,Z -30.583,A -90.000,B 90.000,C 0.000} C_DIS
LIN {X -85.054,Y -23.450,Z -30.521,A -90.000,B 90.000,C 0.000} C_DIS
LIN {X -84.801,Y -23.506,Z -30.450,A -90.000,B 90.000,C 0.000} C_DIS
LIN {X -84.485,Y -23.575,Z -30.374,A -90.000,B 90.000,C 0.000} C_DIS
LIN {X -84.265,Y -23.623,Z -30.329,A -90.000,B 90.000,C 0.000} C_DIS
LIN {X -83.951,Y -23.691,Z -30.275,A -90.000,B 90.000,C 0.000} C_DIS
LIN {X -83.592,Y -23.772,Z -30.225,A -90.000,B 90.000,C 0.000} C_DIS
LIN {X -83.381,Y -23.815,Z -30.202,A -90.000,B 90.000,C 0.000} C_DIS
LIN {X -82.958,Y -23.893,Z -30.171,A -90.000,B 90.000,C 0.000} C_DIS
LIN {X -81.890,Y -24.094,Z -30.105,A -90.000,B 90.000,C 0.000} C_DIS
LIN {X -81.695,Y -24.131,Z -30.095,A -90.000,B 90.000,C 0.000} C_DIS
LIN {X -81.520,Y -24.159,Z -30.086,A -90.000,B 90.000,C 0.000} C_DIS
LIN {X -81.082,Y -24.218,Z -30.075,A -90.000,B 90.000,C 0.000} C_DIS
LIN {X -80.676,Y -24.270,Z -30.082,A -90.000,B 90.000,C 0.000} C_DIS
LIN {X -80.467,Y -24.296,Z -30.092,A -90.000,B 90.000,C 0.000} C_DIS
LIN {X -80.079,Y -24.339,Z -30.119,A -90.000,B 90.000,C 0.000} C_DIS
LIN {X -79.860,Y -24.360,Z -30.138,A -90.000,B 90.000,C 0.000} C_DIS
LIN {X -79.410,Y -24.393,Z -30.193,A -90.000,B 90.000,C 0.000} C_DIS
LIN {X -78.795,Y -24.430,Z -30.284,A -90.000,B 90.000,C 0.000} C_DIS
LIN {X -78.735,Y -24.434,Z -30.293,A -90.000,B 90.000,C 0.000} C_DIS
LIN {X -78.394,Y -24.455,Z -30.345,A -90.000,B 90.000,C 0.000} C_DIS
LIN {X -78.090,Y -24.460,Z -30.392,A -90.000,B 90.000,C 0.000} C_DIS
LIN {X -77.830,Y -24.457,Z -30.432,A -90.000,B 90.000,C 0.000} C_DIS
LIN {X -77.584,Y -24.445,Z -30.475,A -90.000,B 90.000,C 0.000} C_DIS
LIN {X -77.332,Y -24.434,Z -30.526,A -90.000,B 90.000,C 0.000} C_DIS
LIN {X -77.140,Y -24.425,Z -30.571,A -90.000,B 90.000,C 0.000} C_DIS
LIN {X -76.598,Y -24.385,Z -30.710,A -90.000,B 90.000,C 0.000} C_DIS
LIN {X -76.167,Y -24.349,Z -30.832,A -90.000,B 90.000,C 0.000} C_DIS
LIN {X -75.917,Y -24.323,Z -30.904,A -90.000,B 90.000,C 0.000} C_DIS
LIN {X -75.829,Y -24.311,Z -30.929,A -90.000,B 90.000,C 0.000} C_DIS
LIN {X -75.368,Y -24.220,Z -31.061,A -90.000,B 90.000,C 0.000} C_DIS
LIN {X -75.188,Y -24.179,Z -31.113,A -90.000,B 90.000,C 0.000} C_DIS
LIN {X -74.888,Y -24.098,Z -31.202,A -90.000,B 90.000,C 0.000} C_DIS
LIN {X -74.796,Y -24.072,Z -31.230,A -90.000,B 90.000,C 0.000} C_DIS
LIN {X -74.517,Y -23.994,Z -31.325,A -90.000,B 90.000,C 0.000} C_DIS
LIN {X -74.060,Y -23.866,Z -31.486,A -90.000,B 90.000,C 0.000} C_DIS
LIN {X -73.848,Y -23.801,Z -31.561,A -90.000,B 90.000,C 0.000} C_DIS
LIN {X -73.462,Y -23.679,Z -31.699,A -90.000,B 90.000,C 0.000} C_DIS
LIN {X -73.247,Y -23.603,Z -31.776,A -90.000,B 90.000,C 0.000} C_DIS
LIN {X -72.844,Y -23.462,Z -31.911,A -90.000,B 90.000,C 0.000} C_DIS
LIN {X -72.608,Y -23.375,Z -31.991,A -90.000,B 90.000,C 0.000} C_DIS
LIN {X -72.432,Y -23.308,Z -32.054,A -90.000,B 90.000,C 0.000} C_DIS
LIN {X -72.432,Y -60.000,Z -32.054,A -90.000,B 90.000,C 0.000} C_DIS
LIN {X -86.147,Y -60.000,Z -28.775,A -90.000,B 90.000,C 0.000} C_DIS
LIN {X -86.147,Y -23.308,Z -28.775,A -90.000,B 90.000,C 0.000} C_DIS
LIN {X -85.995,Y -23.351,Z -28.723,A -90.000,B 90.000,C 0.000} C_DIS
LIN {X -85.792,Y -23.399,Z -28.656,A -90.000,B 90.000,C 0.000} C_DIS
LIN {X -85.596,Y -23.444,Z -28.596,A -90.000,B 90.000,C 0.000} C_DIS
LIN {X -85.272,Y -23.518,Z -28.506,A -90.000,B 90.000,C 0.000} C_DIS
LIN {X -85.011,Y -23.577,Z -28.443,A -90.000,B 90.000,C 0.000} C_DIS
LIN {X -84.891,Y -23.600,Z -28.416,A -90.000,B 90.000,C 0.000} C_DIS
LIN {X -84.606,Y -23.654,Z -28.358,A -90.000,B 90.000,C 0.000} C_DIS
LIN {X -84.235,Y -23.723,Z -28.296,A -90.000,B 90.000,C 0.000} C_DIS
LIN {X -83.810,Y -23.800,Z -28.237,A -90.000,B 90.000,C 0.000} C_DIS
LIN {X -83.535,Y -23.844,Z -28.209,A -90.000,B 90.000,C 0.000} C_DIS
LIN {X -83.437,Y -23.859,Z -28.201,A -90.000,B 90.000,C 0.000} C_DIS
LIN {X -83.081,Y -23.895,Z -28.175,A -90.000,B 90.000,C 0.000} C_DIS
LIN {X -81.979,Y -24.002,Z -28.109,A -90.000,B 90.000,C 0.000} C_DIS
LIN {X -81.684,Y -24.031,Z -28.095,A -90.000,B 90.000,C 0.000} C_DIS
LIN {X -81.469,Y -24.047,Z -28.088,A -90.000,B 90.000,C 0.000} C_DIS
LIN {X -81.216,Y -24.062,Z -28.083,A -90.000,B 90.000,C 0.000} C_DIS
LIN {X -81.030,Y -24.077,Z -28.081,A -90.000,B 90.000,C 0.000} C_DIS
LIN {X -80.563,Y -24.115,Z -28.091,A -90.000,B 90.000,C 0.000} C_DIS
LIN {X -80.309,Y -24.138,Z -28.104,A -90.000,B 90.000,C 0.000} C_DIS
LIN {X -79.827,Y -24.183,Z -28.140,A -90.000,B 90.000,C 0.000} C_DIS
LIN {X -79.580,Y -24.202,Z -28.164,A -90.000,B 90.000,C 0.000} C_DIS
LIN {X -79.110,Y -24.225,Z -28.223,A -90.000,B 90.000,C 0.000} C_DIS
LIN {X -78.336,Y -24.262,Z -28.339,A -90.000,B 90.000,C 0.000} C_DIS
LIN {X -78.051,Y -24.276,Z -28.382,A -90.000,B 90.000,C 0.000} C_DIS
LIN {X -77.606,Y -24.280,Z -28.451,A -90.000,B 90.000,C 0.000} C_DIS
LIN {X -77.404,Y -24.274,Z -28.484,A -90.000,B 90.000,C 0.000} C_DIS
LIN {X -77.191,Y -24.265,Z -28.523,A -90.000,B 90.000,C 0.000} C_DIS
LIN {X -76.893,Y -24.252,Z -28.583,A -90.000,B 90.000,C 0.000} C_DIS
LIN {X -76.657,Y -24.241,Z -28.639,A -90.000,B 90.000,C 0.000} C_DIS
LIN {X -76.036,Y -24.207,Z -28.799,A -90.000,B 90.000,C 0.000} C_DIS
LIN {X -75.929,Y -24.200,Z -28.829,A -90.000,B 90.000,C 0.000} C_DIS
LIN {X -75.713,Y -24.180,Z -28.890,A -90.000,B 90.000,C 0.000} C_DIS
LIN {X -75.244,Y -24.108,Z -29.026,A -90.000,B 90.000,C 0.000} C_DIS
LIN {X -74.950,Y -24.061,Z -29.108,A -90.000,B 90.000,C 0.000} C_DIS
LIN {X -74.296,Y -23.919,Z -29.300,A -90.000,B 90.000,C 0.000} C_DIS
LIN {X -74.175,Y -23.893,Z -29.337,A -90.000,B 90.000,C 0.000} C_DIS
LIN {X -74.054,Y -23.867,Z -29.378,A -90.000,B 90.000,C 0.000} C_DIS
LIN {X -73.829,Y -23.813,Z -29.455,A -90.000,B 90.000,C 0.000} C_DIS
LIN {X -73.520,Y -23.731,Z -29.563,A -90.000,B 90.000,C 0.000} C_DIS
LIN {X -73.236,Y -23.640,Z -29.664,A -90.000,B 90.000,C 0.000} C_DIS
LIN {X -73.025,Y -23.566,Z -29.740,A -90.000,B 90.000,C 0.000} C_DIS
LIN {X -72.663,Y -23.426,Z -29.871,A -90.000,B 90.000,C 0.000} C_DIS
LIN {X -72.372,Y -23.308,Z -29.970,A -90.000,B 90.000,C 0.000} C_DIS
LIN {X -72.372,Y -60.000,Z -29.970,A -90.000,B 90.000,C 0.000} C_DIS
LIN {X -84.992,Y -60.000,Z -26.426,A -90.000,B 90.000,C 0.000} C_DIS
LIN {X -84.992,Y -23.308,Z -26.426,A -90.000,B 90.000,C 0.000} C_DIS
LIN {X -84.876,Y -23.341,Z -26.401,A -90.000,B 90.000,C 0.000} C_DIS
LIN {X -84.435,Y -23.458,Z -26.324,A -90.000,B 90.000,C 0.000} C_DIS
LIN {X -84.178,Y -23.529,Z -26.285,A -90.000,B 90.000,C 0.000} C_DIS
LIN {X -83.989,Y -23.576,Z -26.258,A -90.000,B 90.000,C 0.000} C_DIS
LIN {X -83.655,Y -23.653,Z -26.221,A -90.000,B 90.000,C 0.000} C_DIS
LIN {X -83.358,Y -23.717,Z -26.197,A -90.000,B 90.000,C 0.000} C_DIS
LIN {X -83.125,Y -23.765,Z -26.178,A -90.000,B 90.000,C 0.000} C_DIS
LIN {X -82.830,Y -23.822,Z -26.159,A -90.000,B 90.000,C 0.000} C_DIS
LIN {X -82.068,Y -23.925,Z -26.113,A -90.000,B 90.000,C 0.000} C_DIS
LIN {X -81.910,Y -23.947,Z -26.105,A -90.000,B 90.000,C 0.000} C_DIS
LIN {X -81.661,Y -23.964,Z -26.094,A -90.000,B 90.000,C 0.000} C_DIS
LIN {X -81.253,Y -23.983,Z -26.085,A -90.000,B 90.000,C 0.000} C_DIS
LIN {X -80.967,Y -23.991,Z -26.083,A -90.000,B 90.000,C 0.000} C_DIS
LIN {X -80.452,Y -24.006,Z -26.097,A -90.000,B 90.000,C 0.000} C_DIS
LIN {X -80.147,Y -24.002,Z -26.115,A -90.000,B 90.000,C 0.000} C_DIS
LIN {X -80.054,Y -24.000,Z -26.123,A -90.000,B 90.000,C 0.000} C_DIS
LIN {X -79.616,Y -23.977,Z -26.162,A -90.000,B 90.000,C 0.000} C_DIS
LIN {X -79.317,Y -23.963,Z -26.196,A -90.000,B 90.000,C 0.000} C_DIS
LIN {X -78.869,Y -23.932,Z -26.259,A -90.000,B 90.000,C 0.000} C_DIS
LIN {X -78.261,Y -23.904,Z -26.358,A -90.000,B 90.000,C 0.000} C_DIS
LIN {X -77.539,Y -23.903,Z -26.474,A -90.000,B 90.000,C 0.000} C_DIS
LIN {X -77.331,Y -23.901,Z -26.506,A -90.000,B 90.000,C 0.000} C_DIS
LIN {X -76.992,Y -23.881,Z -26.566,A -90.000,B 90.000,C 0.000} C_DIS
LIN {X -76.863,Y -23.872,Z -26.589,A -90.000,B 90.000,C 0.000} C_DIS
LIN {X -76.519,Y -23.850,Z -26.660,A -90.000,B 90.000,C 0.000} C_DIS
LIN {X -76.153,Y -23.830,Z -26.747,A -90.000,B 90.000,C 0.000} C_DIS
LIN {X -75.667,Y -23.806,Z -26.872,A -90.000,B 90.000,C 0.000} C_DIS
LIN {X -75.418,Y -23.782,Z -26.941,A -90.000,B 90.000,C 0.000} C_DIS
LIN {X -74.761,Y -23.691,Z -27.130,A -90.000,B 90.000,C 0.000} C_DIS
LIN {X -74.552,Y -23.660,Z -27.188,A -90.000,B 90.000,C 0.000} C_DIS
LIN {X -73.931,Y -23.552,Z -27.365,A -90.000,B 90.000,C 0.000} C_DIS
LIN {X -73.674,Y -23.493,Z -27.443,A -90.000,B 90.000,C 0.000} C_DIS
LIN {X -73.603,Y -23.478,Z -27.466,A -90.000,B 90.000,C 0.000} C_DIS
LIN {X -72.992,Y -23.308,Z -27.681,A -90.000,B 90.000,C 0.000} C_DIS
LIN {X -72.992,Y -60.000,Z -27.681,A -90.000,B 90.000,C 0.000} C_DIS
LIN {X -82.803,Y -60.000,Z -24.225,A -90.000,B 90.000,C 0.000} C_DIS
LIN {X -82.803,Y -23.308,Z -24.225,A -90.000,B 90.000,C 0.000} C_DIS
LIN {X -82.764,Y -23.321,Z -24.221,A -90.000,B 90.000,C 0.000} C_DIS
LIN {X -82.329,Y -23.432,Z -24.181,A -90.000,B 90.000,C 0.000} C_DIS
LIN {X -82.079,Y -23.493,Z -24.160,A -90.000,B 90.000,C 0.000} C_DIS
LIN {X -81.689,Y -23.576,Z -24.133,A -90.000,B 90.000,C 0.000} C_DIS
LIN {X -81.585,Y -23.598,Z -24.127,A -90.000,B 90.000,C 0.000} C_DIS
LIN {X -81.294,Y -23.639,Z -24.115,A -90.000,B 90.000,C 0.000} C_DIS
LIN {X -80.878,Y -23.699,Z -24.107,A -90.000,B 90.000,C 0.000} C_DIS
LIN {X -80.708,Y -23.717,Z -24.109,A -90.000,B 90.000,C 0.000} C_DIS
LIN {X -80.392,Y -23.744,Z -24.115,A -90.000,B 90.000,C 0.000} C_DIS
LIN {X -80.031,Y -23.768,Z -24.132,A -90.000,B 90.000,C 0.000} C_DIS
LIN {X -79.817,Y -23.772,Z -24.149,A -90.000,B 90.000,C 0.000} C_DIS
LIN {X -79.528,Y -23.765,Z -24.174,A -90.000,B 90.000,C 0.000} C_DIS
LIN {X -79.367,Y -23.757,Z -24.189,A -90.000,B 90.000,C 0.000} C_DIS
LIN {X -79.128,Y -23.746,Z -24.217,A -90.000,B 90.000,C 0.000} C_DIS
LIN {X -78.608,Y -23.701,Z -24.290,A -90.000,B 90.000,C 0.000} C_DIS
LIN {X -78.372,Y -23.681,Z -24.329,A -90.000,B 90.000,C 0.000} C_DIS
LIN {X -78.074,Y -23.645,Z -24.380,A -90.000,B 90.000,C 0.000} C_DIS
LIN {X -77.954,Y -23.626,Z -24.402,A -90.000,B 90.000,C 0.000} C_DIS
LIN {X -77.418,Y -23.523,Z -24.504,A -90.000,B 90.000,C 0.000} C_DIS
LIN {X -76.855,Y -23.415,Z -24.618,A -90.000,B 90.000,C 0.000} C_DIS
LIN {X -76.715,Y -23.389,Z -24.647,A -90.000,B 90.000,C 0.000} C_DIS
LIN {X -76.468,Y -23.350,Z -24.699,A -90.000,B 90.000,C 0.000} C_DIS
LIN {X -76.208,Y -23.308,Z -24.760,A -90.000,B 90.000,C 0.000} C_DIS
LIN {X -76.208,Y -60.000,Z -24.760,A -90.000,B 90.000,C 0.000} C_DIS
LIN {X -93.842,Y -60.000,Z -38.730,A -90.000,B 90.000,C 0.000} C_DIS
LIN {X -93.842,Y -23.308,Z -38.730,A -90.000,B 90.000,C 0.000} C_DIS
LIN {X -93.670,Y -23.351,Z -38.714,A -90.000,B 90.000,C 0.000} C_DIS
LIN {X -93.617,Y -23.364,Z -38.710,A -90.000,B 90.000,C 0.000} C_DIS
LIN {X -93.142,Y -23.487,Z -38.690,A -90.000,B 90.000,C 0.000} C_DIS
LIN {X -93.108,Y -23.480,Z -38.629,A -90.000,B 90.000,C 0.000} C_DIS
LIN {X -92.964,Y -23.440,Z -38.397,A -90.000,B 90.000,C 0.000} C_DIS
LIN {X -92.890,Y -23.418,Z -38.284,A -90.000,B 90.000,C 0.000} C_DIS
LIN {X -92.766,Y -23.385,Z -38.102,A -90.000,B 90.000,C 0.000} C_DIS
LIN {X -92.651,Y -23.366,Z -37.946,A -90.000,B 90.000,C 0.000} C_DIS
LIN {X -92.596,Y -23.350,Z -37.852,A -90.000,B 90.000,C 0.000} C_DIS
LIN {X -92.517,Y -23.330,Z -37.723,A -90.000,B 90.000,C 0.000} C_DIS
LIN {X -92.458,Y -23.308,Z -37.633,A -90.000,B 90.000,C 0.000} C_DIS
LIN {X -92.458,Y -60.000,Z -37.633,A -90.000,B 90.000,C 0.000} C_DIS
LIN {X -103.472,Y -60.000,Z -48.295,A -90.000,B 90.000,C 0.000} C_DIS
LIN {X -103.472,Y -23.308,Z -48.295,A -90.000,B 90.000,C 0.000} C_DIS
LIN {X -103.511,Y -23.351,Z -48.034,A -90.000,B 90.000,C 0.000} C_DIS
LIN {X -103.532,Y -23.390,Z -47.824,A -90.000,B 90.000,C 0.000} C_DIS
LIN {X -103.541,Y -23.433,Z -47.505,A -90.000,B 90.000,C 0.000} C_DIS
LIN {X -103.545,Y -23.464,Z -47.257,A -90.000,B 90.000,C 0.000} C_DIS
LIN {X -103.543,Y -23.484,Z -47.116,A -90.000,B 90.000,C 0.000} C_DIS
LIN {X -103.533,Y -23.509,Z -46.953,A -90.000,B 90.000,C 0.000} C_DIS
LIN {X -103.520,Y -23.536,Z -46.799,A -90.000,B 90.000,C 0.000} C_DIS
LIN {X -103.479,Y -23.573,Z -46.489,A -90.000,B 90.000,C 0.000} C_DIS
LIN {X -103.426,Y -23.608,Z -46.158,A -90.000,B 90.000,C 0.000} C_DIS
LIN {X -103.390,Y -23.620,Z -45.977,A -90.000,B 90.000,C 0.000} C_DIS
LIN {X -103.345,Y -23.635,Z -45.801,A -90.000,B 90.000,C 0.000} C_DIS
LIN {X -103.318,Y -23.641,Z -45.703,A -90.000,B 90.000,C 0.000} C_DIS
LIN {X -103.238,Y -23.662,Z -45.467,A -90.000,B 90.000,C 0.000} C_DIS
LIN {X -103.182,Y -23.677,Z -45.316,A -90.000,B 90.000,C 0.000} C_DIS
LIN {X -103.093,Y -23.693,Z -45.091,A -90.000,B 90.000,C 0.000} C_DIS
LIN {X -103.068,Y -23.698,Z -45.033,A -90.000,B 90.000,C 0.000} C_DIS
LIN {X -102.922,Y -23.707,Z -44.717,A -90.000,B 90.000,C 0.000} C_DIS
LIN {X -102.832,Y -23.713,Z -44.536,A -90.000,B 90.000,C 0.000} C_DIS
LIN {X -102.780,Y -23.718,Z -44.440,A -90.000,B 90.000,C 0.000} C_DIS
LIN {X -102.668,Y -23.717,Z -44.261,A -90.000,B 90.000,C 0.000} C_DIS
LIN {X -102.549,Y -23.718,Z -44.077,A -90.000,B 90.000,C 0.000} C_DIS
LIN {X -102.411,Y -23.721,Z -43.874,A -90.000,B 90.000,C 0.000} C_DIS
LIN {X -102.211,Y -23.715,Z -43.627,A -90.000,B 90.000,C 0.000} C_DIS
LIN {X -102.019,Y -23.707,Z -43.396,A -90.000,B 90.000,C 0.000} C_DIS
LIN {X -101.968,Y -23.707,Z -43.338,A -90.000,B 90.000,C 0.000} C_DIS
LIN {X -101.738,Y -23.689,Z -43.101,A -90.000,B 90.000,C 0.000} C_DIS
LIN {X -101.597,Y -23.673,Z -42.964,A -90.000,B 90.000,C 0.000} C_DIS
LIN {X -101.490,Y -23.665,Z -42.868,A -90.000,B 90.000,C 0.000} C_DIS
LIN {X -101.347,Y -23.655,Z -42.750,A -90.000,B 90.000,C 0.000} C_DIS
LIN {X -101.168,Y -23.639,Z -42.612,A -90.000,B 90.000,C 0.000} C_DIS
LIN {X -101.069,Y -23.626,Z -42.531,A -90.000,B 90.000,C 0.000} C_DIS
LIN {X -100.912,Y -23.602,Z -42.420,A -90.000,B 90.000,C 0.000} C_DIS
LIN {X -100.581,Y -23.550,Z -42.203,A -90.000,B 90.000,C 0.000} C_DIS
LIN {X -100.477,Y -23.535,Z -42.136,A -90.000,B 90.000,C 0.000} C_DIS
LIN {X -100.344,Y -23.517,Z -42.056,A -90.000,B 90.000,C 0.000} C_DIS
LIN {X -100.304,Y -23.512,Z -42.034,A -90.000,B 90.000,C 0.000} C_DIS
LIN {X -100.054,Y -23.467,Z -41.909,A -90.000,B 90.000,C 0.000} C_DIS
LIN {X -99.879,Y -23.431,Z -41.829,A -90.000,B 90.000,C 0.000} C_DIS
LIN {X -99.711,Y -23.400,Z -41.756,A -90.000,B 90.000,C 0.000} C_DIS
LIN {X -99.518,Y -23.369,Z -41.679,A -90.000,B 90.000,C 0.000} C_DIS
LIN {X -99.272,Y -23.322,Z -41.577,A -90.000,B 90.000,C 0.000} C_DIS
LIN {X -99.196,Y -23.308,Z -41.548,A -90.000,B 90.000,C 0.000} C_DIS
LIN {X -99.196,Y -60.000,Z -41.548,A -90.000,B 90.000,C 0.000} C_DIS
LIN {X -97.971,Y -60.000,Z -60.610,A -90.000,B 90.000,C 0.000} C_DIS
LIN {X -97.971,Y -23.308,Z -60.610,A -90.000,B 90.000,C 0.000} C_DIS
LIN {X -98.151,Y -23.361,Z -60.357,A -90.000,B 90.000,C 0.000} C_DIS
LIN {X -98.250,Y -23.382,Z -60.230,A -90.000,B 90.000,C 0.000} C_DIS
LIN {X -98.400,Y -23.405,Z -60.023,A -90.000,B 90.000,C 0.000} C_DIS
LIN {X -98.603,Y -23.440,Z -59.732,A -90.000,B 90.000,C 0.000} C_DIS
LIN {X -98.675,Y -23.456,Z -59.624,A -90.000,B 90.000,C 0.000} C_DIS
LIN {X -98.889,Y -23.508,Z -59.284,A -90.000,B 90.000,C 0.000} C_DIS
LIN {X -99.026,Y -23.538,Z -59.061,A -90.000,B 90.000,C 0.000} C_DIS
LIN {X -99.274,Y -23.590,Z -58.656,A -90.000,B 90.000,C 0.000} C_DIS
LIN {X -99.317,Y -23.595,Z -58.581,A -90.000,B 90.000,C 0.000} C_DIS
LIN {X -99.371,Y -23.604,Z -58.481,A -90.000,B 90.000,C 0.000} C_DIS
LIN {X -99.456,Y -23.620,Z -58.313,A -90.000,B 90.000,C 0.000} C_DIS
LIN {X -99.596,Y -23.652,Z -58.021,A -90.000,B 90.000,C 0.000} C_DIS
LIN {X -99.733,Y -23.676,Z -57.723,A -90.000,B 90.000,C 0.000} C_DIS
LIN {X -99.781,Y -23.688,Z -57.610,A -90.000,B 90.000,C 0.000} C_DIS
LIN {X -99.827,Y -23.697,Z -57.491,A -90.000,B 90.000,C 0.000} C_DIS
LIN {X -99.948,Y -23.726,Z -57.158,A -90.000,B 90.000,C 0.000} C_DIS
LIN {X -100.001,Y -23.744,Z -56.992,A -90.000,B 90.000,C 0.000} C_DIS
LIN {X -100.031,Y -23.755,Z -56.883,A -90.000,B 90.000,C 0.000} C_DIS
LIN {X -100.063,Y -23.769,Z -56.754,A -90.000,B 90.000,C 0.000} C_DIS
LIN {X -100.121,Y -23.790,Z -56.504,A -90.000,B 90.000,C 0.000} C_DIS
LIN {X -100.172,Y -23.816,Z -56.242,A -90.000,B 90.000,C 0.000} C_DIS
LIN {X -100.210,Y -23.839,Z -56.014,A -90.000,B 90.000,C 0.000} C_DIS
LIN {X -100.222,Y -23.846,Z -55.918,A -90.000,B 90.000,C 0.000} C_DIS
LIN {X -100.383,Y -23.800,Z -55.685,A -90.000,B 90.000,C 0.000} C_DIS
LIN {X -100.497,Y -23.765,Z -55.514,A -90.000,B 90.000,C 0.000} C_DIS
LIN {X -100.645,Y -23.720,Z -55.281,A -90.000,B 90.000,C 0.000} C_DIS
LIN {X -100.790,Y -23.676,Z -55.045,A -90.000,B 90.000,C 0.000} C_DIS
LIN {X -100.897,Y -23.637,Z -54.859,A -90.000,B 90.000,C 0.000} C_DIS
LIN {X -101.046,Y -23.574,Z -54.586,A -90.000,B 90.000,C 0.000} C_DIS
LIN {X -101.160,Y -23.526,Z -54.366,A -90.000,B 90.000,C 0.000} C_DIS
LIN {X -101.242,Y -23.486,Z -54.200,A -90.000,B 90.000,C 0.000} C_DIS
LIN {X -101.306,Y -23.454,Z -54.061,A -90.000,B 90.000,C 0.000} C_DIS
LIN {X -101.346,Y -23.434,Z -53.968,A -90.000,B 90.000,C 0.000} C_DIS
LIN {X -101.427,Y -23.392,Z -53.763,A -90.000,B 90.000,C 0.000} C_DIS
LIN {X -101.574,Y -23.308,Z -53.513,A -90.000,B 90.000,C 0.000} C_DIS
LIN {X -101.574,Y -60.000,Z -53.513,A -90.000,B 90.000,C 0.000} C_DIS
LIN {X -105.623,Y -60.000,Z -243.561,A -90.000,B 90.000,C 0.000} C_DIS
LIN {X -105.623,Y -23.308,Z -243.561,A -90.000,B 90.000,C 0.000} C_DIS
LIN {X -102.579,Y -23.308,Z -241.509,A -90.000,B 90.000,C 0.000} C_DIS
LIN {X -102.258,Y -23.308,Z -241.299,A -90.000,B 90.000,C 0.000} C_DIS
LIN {X -94.671,Y -23.308,Z -236.287,A -90.000,B 90.000,C 0.000} C_DIS
LIN {X -86.436,Y -23.308,Z -230.982,A -90.000,B 90.000,C 0.000} C_DIS
LIN {X -78.058,Y -23.308,Z -225.744,A -90.000,B 90.000,C 0.000} C_DIS
LIN {X -70.407,Y -23.308,Z -221.136,A -90.000,B 90.000,C 0.000} C_DIS
LIN {X -69.401,Y -23.308,Z -220.532,A -90.000,B 90.000,C 0.000} C_DIS
LIN {X -69.035,Y -23.308,Z -220.315,A -90.000,B 90.000,C 0.000} C_DIS
LIN {X -62.034,Y -23.308,Z -216.202,A -90.000,B 90.000,C 0.000} C_DIS
LIN {X -59.725,Y -23.308,Z -214.857,A -90.000,B 90.000,C 0.000} C_DIS
LIN {X -59.360,Y -23.308,Z -214.644,A -90.000,B 90.000,C 0.000} C_DIS
LIN {X -52.900,Y -23.308,Z -210.900,A -90.000,B 90.000,C 0.000} C_DIS
LIN {X -51.892,Y -23.308,Z -210.305,A -90.000,B 90.000,C 0.000} C_DIS
LIN {X -45.910,Y -23.308,Z -206.843,A -90.000,B 90.000,C 0.000} C_DIS
LIN {X -42.712,Y -23.308,Z -204.958,A -90.000,B 90.000,C 0.000} C_DIS
LIN {X -39.350,Y -23.308,Z -202.913,A -90.000,B 90.000,C 0.000} C_DIS
LIN {X -37.993,Y -23.308,Z -202.052,A -90.000,B 90.000,C 0.000} C_DIS
LIN {X -37.215,Y -23.308,Z -201.531,A -90.000,B 90.000,C 0.000} C_DIS
LIN {X -36.268,Y -23.308,Z -200.851,A -90.000,B 90.000,C 0.000} C_DIS
LIN {X -35.341,Y -23.308,Z -200.178,A -90.000,B 90.000,C 0.000} C_DIS
LIN {X -32.882,Y -23.308,Z -198.217,A -90.000,B 90.000,C 0.000} C_DIS
LIN {X -31.008,Y -23.308,Z -196.620,A -90.000,B 90.000,C 0.000} C_DIS
LIN {X -29.667,Y -23.308,Z -195.495,A -90.000,B 90.000,C 0.000} C_DIS
LIN {X -26.664,Y -23.308,Z -192.944,A -90.000,B 90.000,C 0.000} C_DIS
LIN {X -26.071,Y -23.308,Z -192.420,A -90.000,B 90.000,C 0.000} C_DIS
LIN {X -23.825,Y -23.308,Z -190.470,A -90.000,B 90.000,C 0.000} C_DIS
LIN {X -23.428,Y -23.308,Z -190.096,A -90.000,B 90.000,C 0.000} C_DIS
LIN {X -21.210,Y -23.308,Z -188.067,A -90.000,B 90.000,C 0.000} C_DIS
LIN {X -20.343,Y -23.308,Z -187.184,A -90.000,B 90.000,C 0.000} C_DIS
LIN {X -18.629,Y -23.308,Z -185.485,A -90.000,B 90.000,C 0.000} C_DIS
LIN {X -16.677,Y -23.308,Z -183.344,A -90.000,B 90.000,C 0.000} C_DIS
LIN {X -16.126,Y -23.308,Z -182.724,A -90.000,B 90.000,C 0.000} C_DIS
LIN {X -14.104,Y -23.308,Z -180.248,A -90.000,B 90.000,C 0.000} C_DIS
LIN {X -13.812,Y -23.308,Z -179.882,A -90.000,B 90.000,C 0.000} C_DIS
LIN {X -11.599,Y -23.308,Z -176.796,A -90.000,B 90.000,C 0.000} C_DIS
LIN {X -11.536,Y -23.308,Z -176.694,A -90.000,B 90.000,C 0.000} C_DIS
LIN {X -9.733,Y -23.308,Z -173.767,A -90.000,B 90.000,C 0.000} C_DIS
LIN {X -9.643,Y -23.308,Z -173.603,A -90.000,B 90.000,C 0.000} C_DIS
LIN {X -8.150,Y -23.308,Z -170.611,A -90.000,B 90.000,C 0.000} C_DIS
LIN {X -7.018,Y -23.308,Z -167.585,A -90.000,B 90.000,C 0.000} C_DIS
LIN {X -6.758,Y -23.308,Z -166.447,A -90.000,B 90.000,C 0.000} C_DIS
LIN {X -6.392,Y -23.308,Z -164.883,A -90.000,B 90.000,C 0.000} C_DIS
LIN {X -6.294,Y -23.308,Z -162.869,A -90.000,B 90.000,C 0.000} C_DIS
LIN {X -6.561,Y -23.308,Z -161.785,A -90.000,B 90.000,C 0.000} C_DIS
LIN {X -6.614,Y -23.308,Z -161.526,A -90.000,B 90.000,C 0.000} C_DIS
LIN {X -6.938,Y -23.308,Z -160.970,A -90.000,B 90.000,C 0.000} C_DIS
LIN {X -7.178,Y -23.308,Z -160.502,A -90.000,B 90.000,C 0.000} C_DIS
LIN {X -7.549,Y -23.308,Z -160.102,A -90.000,B 90.000,C 0.000} C_DIS
LIN {X -8.034,Y -23.308,Z -159.527,A -90.000,B 90.000,C 0.000} C_DIS
LIN {X -8.331,Y -23.308,Z -159.279,A -90.000,B 90.000,C 0.000} C_DIS
LIN {X -9.460,Y -23.308,Z -158.247,A -90.000,B 90.000,C 0.000} C_DIS
LIN {X -10.702,Y -23.308,Z -157.194,A -90.000,B 90.000,C 0.000} C_DIS
LIN {X -11.064,Y -23.308,Z -156.876,A -90.000,B 90.000,C 0.000} C_DIS
LIN {X -12.479,Y -23.308,Z -155.691,A -90.000,B 90.000,C 0.000} C_DIS
LIN {X -12.827,Y -23.308,Z -155.394,A -90.000,B 90.000,C 0.000} C_DIS
LIN {X -12.979,Y -23.308,Z -155.261,A -90.000,B 90.000,C 0.000} C_DIS
LIN {X -14.516,Y -23.308,Z -153.994,A -90.000,B 90.000,C 0.000} C_DIS
LIN {X -14.861,Y -23.308,Z -153.704,A -90.000,B 90.000,C 0.000} C_DIS
LIN {X -15.126,Y -23.308,Z -153.475,A -90.000,B 90.000,C 0.000} C_DIS
LIN {X -16.984,Y -23.308,Z -151.939,A -90.000,B 90.000,C 0.000} C_DIS
LIN {X -17.335,Y -23.308,Z -151.643,A -90.000,B 90.000,C 0.000} C_DIS
LIN {X -17.935,Y -23.308,Z -151.130,A -90.000,B 90.000,C 0.000} C_DIS
LIN {X -20.316,Y -23.308,Z -149.130,A -90.000,B 90.000,C 0.000} C_DIS
LIN {X -20.890,Y -23.308,Z -148.609,A -90.000,B 90.000,C 0.000} C_DIS
LIN {X -23.557,Y -23.308,Z -146.200,A -90.000,B 90.000,C 0.000} C_DIS
LIN {X -26.406,Y -23.308,Z -143.286,A -90.000,B 90.000,C 0.000} C_DIS
LIN {X -26.848,Y -23.308,Z -142.830,A -90.000,B 90.000,C 0.000} C_DIS
LIN {X -27.119,Y -23.308,Z -142.548,A -90.000,B 90.000,C 0.000} C_DIS
LIN {X -28.995,Y -23.308,Z -140.244,A -90.000,B 90.000,C 0.000} C_DIS
LIN {X -30.113,Y -23.308,Z -138.860,A -90.000,B 90.000,C 0.000} C_DIS
LIN {X -30.373,Y -23.308,Z -138.522,A -90.000,B 90.000,C 0.000} C_DIS
LIN {X -30.747,Y -23.308,Z -137.924,A -90.000,B 90.000,C 0.000} C_DIS
LIN {X -31.827,Y -23.308,Z -136.199,A -90.000,B 90.000,C 0.000} C_DIS
LIN {X -32.887,Y -23.308,Z -134.570,A -90.000,B 90.000,C 0.000} C_DIS
LIN {X -33.314,Y -23.308,Z -134.051,A -90.000,B 90.000,C 0.000} C_DIS
LIN {X -33.675,Y -23.308,Z -133.520,A -90.000,B 90.000,C 0.000} C_DIS
LIN {X -35.907,Y -23.308,Z -130.179,A -90.000,B 90.000,C 0.000} C_DIS
LIN {X -38.126,Y -23.308,Z -126.127,A -90.000,B 90.000,C 0.000} C_DIS
LIN {X -38.234,Y -23.308,Z -125.927,A -90.000,B 90.000,C 0.000} C_DIS
LIN {X -38.830,Y -23.308,Z -124.589,A -90.000,B 90.000,C 0.000} C_DIS
LIN {X -39.763,Y -23.308,Z -122.731,A -90.000,B 90.000,C 0.000} C_DIS
LIN {X -40.431,Y -23.308,Z -121.313,A -90.000,B 90.000,C 0.000} C_DIS
LIN {X -40.748,Y -23.308,Z -120.597,A -90.000,B 90.000,C 0.000} C_DIS
LIN {X -41.499,Y -23.308,Z -119.091,A -90.000,B 90.000,C 0.000} C_DIS
LIN {X -41.673,Y -23.308,Z -118.684,A -90.000,B 90.000,C 0.000} C_DIS
LIN {X -42.519,Y -23.308,Z -117.142,A -90.000,B 90.000,C 0.000} C_DIS
LIN {X -42.563,Y -23.308,Z -117.051,A -90.000,B 90.000,C 0.000} C_DIS
LIN {X -43.660,Y -23.308,Z -115.319,A -90.000,B 90.000,C 0.000} C_DIS
LIN {X -45.370,Y -23.308,Z -112.891,A -90.000,B 90.000,C 0.000} C_DIS
LIN {X -46.950,Y -23.308,Z -110.741,A -90.000,B 90.000,C 0.000} C_DIS
LIN {X -47.636,Y -23.308,Z -109.813,A -90.000,B 90.000,C 0.000} C_DIS
LIN {X -48.567,Y -23.308,Z -108.571,A -90.000,B 90.000,C 0.000} C_DIS
LIN {X -50.467,Y -23.308,Z -106.100,A -90.000,B 90.000,C 0.000} C_DIS
LIN {X -51.806,Y -23.308,Z -104.321,A -90.000,B 90.000,C 0.000} C_DIS
LIN {X -52.395,Y -23.308,Z -103.571,A -90.000,B 90.000,C 0.000} C_DIS
LIN {X -52.665,Y -23.308,Z -103.221,A -90.000,B 90.000,C 0.000} C_DIS
LIN {X -53.590,Y -23.308,Z -101.969,A -90.000,B 90.000,C 0.000} C_DIS
LIN {X -55.150,Y -23.308,Z -99.940,A -90.000,B 90.000,C 0.000} C_DIS
LIN {X -55.493,Y -23.308,Z -99.485,A -90.000,B 90.000,C 0.000} C_DIS
LIN {X -56.888,Y -23.308,Z -97.598,A -90.000,B 90.000,C 0.000} C_DIS
LIN {X -57.507,Y -23.308,Z -96.790,A -90.000,B 90.000,C 0.000} C_DIS
LIN {X -58.501,Y -23.308,Z -95.455,A -90.000,B 90.000,C 0.000} C_DIS
LIN {X -59.682,Y -23.308,Z -93.921,A -90.000,B 90.000,C 0.000} C_DIS
LIN {X -60.267,Y -23.308,Z -93.176,A -90.000,B 90.000,C 0.000} C_DIS
LIN {X -60.902,Y -23.308,Z -92.364,A -90.000,B 90.000,C 0.000} C_DIS
LIN {X -61.081,Y -23.308,Z -92.131,A -90.000,B 90.000,C 0.000} C_DIS
LIN {X -61.479,Y -23.308,Z -91.609,A -90.000,B 90.000,C 0.000} C_DIS
LIN {X -61.587,Y -23.308,Z -91.473,A -90.000,B 90.000,C 0.000} C_DIS
LIN {X -61.924,Y -23.308,Z -91.068,A -90.000,B 90.000,C 0.000} C_DIS
LIN {X -63.495,Y -23.308,Z -89.130,A -90.000,B 90.000,C 0.000} C_DIS
LIN {X -64.536,Y -23.308,Z -87.945,A -90.000,B 90.000,C 0.000} C_DIS
LIN {X -65.319,Y -23.308,Z -87.030,A -90.000,B 90.000,C 0.000} C_DIS
LIN {X -66.944,Y -23.308,Z -85.261,A -90.000,B 90.000,C 0.000} C_DIS
LIN {X -67.089,Y -23.308,Z -85.100,A -90.000,B 90.000,C 0.000} C_DIS
LIN {X -67.484,Y -23.308,Z -84.681,A -90.000,B 90.000,C 0.000} C_DIS
LIN {X -68.838,Y -23.308,Z -83.218,A -90.000,B 90.000,C 0.000} C_DIS
LIN {X -69.492,Y -23.308,Z -82.529,A -90.000,B 90.000,C 0.000} C_DIS
LIN {X -70.506,Y -23.308,Z -81.441,A -90.000,B 90.000,C 0.000} C_DIS
LIN {X -72.011,Y -23.308,Z -79.891,A -90.000,B 90.000,C 0.000} C_DIS
LIN {X -72.390,Y -23.308,Z -79.519,A -90.000,B 90.000,C 0.000} C_DIS
LIN {X -73.541,Y -23.308,Z -78.359,A -90.000,B 90.000,C 0.000} C_DIS
LIN {X -74.624,Y -23.308,Z -77.383,A -90.000,B 90.000,C 0.000} C_DIS
LIN {X -75.099,Y -23.308,Z -77.050,A -90.000,B 90.000,C 0.000} C_DIS
LIN {X -75.420,Y -23.308,Z -77.008,A -90.000,B 90.000,C 0.000} C_DIS
LIN {X -75.477,Y -23.308,Z -76.999,A -90.000,B 90.000,C 0.000} C_DIS
LIN {X -75.548,Y -23.308,Z -76.994,A -90.000,B 90.000,C 0.000} C_DIS
LIN {X -75.892,Y -23.308,Z -76.960,A -90.000,B 90.000,C 0.000} C_DIS
LIN {X -76.238,Y -23.308,Z -76.956,A -90.000,B 90.000,C 0.000} C_DIS
LIN {X -76.378,Y -23.308,Z -76.953,A -90.000,B 90.000,C 0.000} C_DIS
LIN {X -76.750,Y -23.308,Z -76.935,A -90.000,B 90.000,C 0.000} C_DIS
LIN {X -76.830,Y -23.308,Z -76.926,A -90.000,B 90.000,C 0.000} C_DIS
LIN {X -77.198,Y -23.308,Z -76.867,A -90.000,B 90.000,C 0.000} C_DIS
LIN {X -77.323,Y -23.308,Z -76.839,A -90.000,B 90.000,C 0.000} C_DIS
LIN {X -77.970,Y -23.308,Z -76.668,A -90.000,B 90.000,C 0.000} C_DIS
LIN {X -78.495,Y -23.308,Z -76.538,A -90.000,B 90.000,C 0.000} C_DIS
LIN {X -78.974,Y -23.308,Z -76.406,A -90.000,B 90.000,C 0.000} C_DIS
LIN {X -79.049,Y -23.308,Z -76.384,A -90.000,B 90.000,C 0.000} C_DIS
LIN {X -79.295,Y -23.308,Z -76.295,A -90.000,B 90.000,C 0.000} C_DIS
LIN {X -79.867,Y -23.308,Z -76.068,A -90.000,B 90.000,C 0.000} C_DIS
LIN {X -80.638,Y -23.308,Z -75.684,A -90.000,B 90.000,C 0.000} C_DIS
LIN {X -81.041,Y -23.308,Z -75.471,A -90.000,B 90.000,C 0.000} C_DIS
LIN {X -82.000,Y -23.308,Z -74.890,A -90.000,B 90.000,C 0.000} C_DIS
LIN {X -82.489,Y -23.308,Z -74.559,A -90.000,B 90.000,C 0.000} C_DIS
LIN {X -82.562,Y -23.308,Z -74.506,A -90.000,B 90.000,C 0.000} C_DIS
LIN {X -83.532,Y -23.308,Z -73.714,A -90.000,B 90.000,C 0.000} C_DIS
LIN {X -83.878,Y -23.308,Z -73.419,A -90.000,B 90.000,C 0.000} C_DIS
LIN {X -84.103,Y -23.308,Z -73.196,A -90.000,B 90.000,C 0.000} C_DIS
LIN {X -84.808,Y -23.308,Z -72.453,A -90.000,B 90.000,C 0.000} C_DIS
LIN {X -84.981,Y -23.308,Z -72.269,A -90.000,B 90.000,C 0.000} C_DIS
LIN {X -85.161,Y -23.308,Z -72.065,A -90.000,B 90.000,C 0.000} C_DIS
LIN {X -85.200,Y -23.308,Z -72.024,A -90.000,B 90.000,C 0.000} C_DIS
LIN {X -85.547,Y -23.308,Z -71.573,A -90.000,B 90.000,C 0.000} C_DIS
LIN {X -85.748,Y -23.308,Z -71.308,A -90.000,B 90.000,C 0.000} C_DIS
LIN {X -86.188,Y -23.308,Z -70.823,A -90.000,B 90.000,C 0.000} C_DIS
LIN {X -86.488,Y -23.308,Z -70.517,A -90.000,B 90.000,C 0.000} C_DIS
LIN {X -86.593,Y -23.308,Z -70.423,A -90.000,B 90.000,C 0.000} C_DIS
LIN {X -87.055,Y -23.308,Z -69.977,A -90.000,B 90.000,C 0.000} C_DIS
LIN {X -87.294,Y -23.308,Z -69.761,A -90.000,B 90.000,C 0.000} C_DIS
LIN {X -87.633,Y -23.308,Z -69.445,A -90.000,B 90.000,C 0.000} C_DIS
LIN {X -87.826,Y -23.308,Z -69.244,A -90.000,B 90.000,C 0.000} C_DIS
LIN {X -88.186,Y -23.308,Z -68.903,A -90.000,B 90.000,C 0.000} C_DIS
LIN {X -88.310,Y -23.308,Z -68.774,A -90.000,B 90.000,C 0.000} C_DIS
LIN {X -88.774,Y -23.308,Z -68.330,A -90.000,B 90.000,C 0.000} C_DIS
LIN {X -89.376,Y -23.308,Z -67.776,A -90.000,B 90.000,C 0.000} C_DIS
LIN {X -89.949,Y -23.308,Z -67.289,A -90.000,B 90.000,C 0.000} C_DIS
LIN {X -90.687,Y -23.308,Z -66.724,A -90.000,B 90.000,C 0.000} C_DIS
LIN {X -91.532,Y -23.308,Z -66.101,A -90.000,B 90.000,C 0.000} C_DIS
LIN {X -92.710,Y -23.308,Z -65.227,A -90.000,B 90.000,C 0.000} C_DIS
LIN {X -93.660,Y -23.308,Z -64.486,A -90.000,B 90.000,C 0.000} C_DIS
LIN {X -93.739,Y -23.308,Z -64.423,A -90.000,B 90.000,C 0.000} C_DIS
LIN {X -94.598,Y -23.308,Z -63.680,A -90.000,B 90.000,C 0.000} C_DIS
LIN {X -95.588,Y -23.308,Z -62.769,A -90.000,B 90.000,C 0.000} C_DIS
LIN {X -95.919,Y -23.308,Z -62.461,A -90.000,B 90.000,C 0.000} C_DIS
LIN {X -96.257,Y -23.308,Z -62.142,A -90.000,B 90.000,C 0.000} C_DIS
LIN {X -96.753,Y -23.308,Z -61.687,A -90.000,B 90.000,C 0.000} C_DIS
LIN {X -97.107,Y -23.308,Z -61.368,A -90.000,B 90.000,C 0.000} C_DIS
LIN {X -97.636,Y -23.308,Z -60.921,A -90.000,B 90.000,C 0.000} C_DIS
LIN {X -98.497,Y -23.308,Z -60.120,A -90.000,B 90.000,C 0.000} C_DIS
LIN {X -99.056,Y -23.308,Z -59.521,A -90.000,B 90.000,C 0.000} C_DIS
LIN {X -99.633,Y -23.308,Z -58.872,A -90.000,B 90.000,C 0.000} C_DIS
LIN {X -99.795,Y -23.308,Z -58.683,A -90.000,B 90.000,C 0.000} C_DIS
LIN {X -100.083,Y -23.308,Z -58.296,A -90.000,B 90.000,C 0.000} C_DIS
LIN {X -100.289,Y -23.308,Z -58.011,A -90.000,B 90.000,C 0.000} C_DIS
LIN {X -100.612,Y -23.308,Z -57.495,A -90.000,B 90.000,C 0.000} C_DIS
LIN {X -100.880,Y -23.308,Z -56.984,A -90.000,B 90.000,C 0.000} C_DIS
LIN {X -100.957,Y -23.308,Z -56.830,A -90.000,B 90.000,C 0.000} C_DIS
LIN {X -101.243,Y -23.308,Z -56.091,A -90.000,B 90.000,C 0.000} C_DIS
LIN {X -101.272,Y -23.308,Z -56.013,A -90.000,B 90.000,C 0.000} C_DIS
LIN {X -101.373,Y -23.308,Z -55.705,A -90.000,B 90.000,C 0.000} C_DIS
LIN {X -101.485,Y -23.308,Z -55.219,A -90.000,B 90.000,C 0.000} C_DIS
LIN {X -101.520,Y -23.308,Z -55.065,A -90.000,B 90.000,C 0.000} C_DIS
LIN {X -101.559,Y -23.308,Z -54.838,A -90.000,B 90.000,C 0.000} C_DIS
LIN {X -101.606,Y -23.308,Z -54.412,A -90.000,B 90.000,C 0.000} C_DIS
LIN {X -101.626,Y -23.308,Z -54.112,A -90.000,B 90.000,C 0.000} C_DIS
LIN {X -101.622,Y -23.308,Z -54.018,A -90.000,B 90.000,C 0.000} C_DIS
LIN {X -101.593,Y -23.308,Z -53.700,A -90.000,B 90.000,C 0.000} C_DIS
LIN {X -101.555,Y -23.308,Z -53.327,A -90.000,B 90.000,C 0.000} C_DIS
LIN {X -101.477,Y -23.308,Z -53.017,A -90.000,B 90.000,C 0.000} C_DIS
LIN {X -101.352,Y -23.308,Z -52.723,A -90.000,B 90.000,C 0.000} C_DIS
LIN {X -101.182,Y -23.308,Z -52.453,A -90.000,B 90.000,C 0.000} C_DIS
LIN {X -101.114,Y -23.308,Z -52.356,A -90.000,B 90.000,C 0.000} C_DIS
LIN {X -100.985,Y -23.308,Z -52.154,A -90.000,B 90.000,C 0.000} C_DIS
LIN {X -101.291,Y -23.308,Z -51.803,A -90.000,B 90.000,C 0.000} C_DIS
LIN {X -101.562,Y -23.308,Z -51.478,A -90.000,B 90.000,C 0.000} C_DIS
LIN {X -101.720,Y -23.308,Z -51.278,A -90.000,B 90.000,C 0.000} C_DIS
LIN {X -102.595,Y -23.308,Z -49.996,A -90.000,B 90.000,C 0.000} C_DIS
LIN {X -102.990,Y -23.308,Z -49.304,A -90.000,B 90.000,C 0.000} C_DIS
LIN {X -103.193,Y -23.308,Z -48.929,A -90.000,B 90.000,C 0.000} C_DIS
LIN {X -103.333,Y -23.308,Z -48.665,A -90.000,B 90.000,C 0.000} C_DIS
LIN {X -103.365,Y -23.308,Z -48.586,A -90.000,B 90.000,C 0.000} C_DIS
LIN {X -103.516,Y -23.308,Z -48.177,A -90.000,B 90.000,C 0.000} C_DIS
LIN {X -103.668,Y -23.308,Z -47.746,A -90.000,B 90.000,C 0.000} C_DIS
LIN {X -103.751,Y -23.308,Z -47.376,A -90.000,B 90.000,C 0.000} C_DIS
LIN {X -103.831,Y -23.308,Z -46.977,A -90.000,B 90.000,C 0.000} C_DIS
LIN {X -103.909,Y -23.308,Z -46.541,A -90.000,B 90.000,C 0.000} C_DIS
LIN {X -103.929,Y -23.308,Z -46.190,A -90.000,B 90.000,C 0.000} C_DIS
LIN {X -103.936,Y -23.308,Z -45.821,A -90.000,B 90.000,C 0.000} C_DIS
LIN {X -103.907,Y -23.308,Z -45.471,A -90.000,B 90.000,C 0.000} C_DIS
LIN {X -103.873,Y -23.308,Z -45.248,A -90.000,B 90.000,C 0.000} C_DIS
LIN {X -103.811,Y -23.308,Z -44.908,A -90.000,B 90.000,C 0.000} C_DIS
LIN {X -103.733,Y -23.308,Z -44.598,A -90.000,B 90.000,C 0.000} C_DIS
LIN {X -103.606,Y -23.308,Z -44.282,A -90.000,B 90.000,C 0.000} C_DIS
LIN {X -103.480,Y -23.308,Z -43.988,A -90.000,B 90.000,C 0.000} C_DIS
LIN {X -103.180,Y -23.308,Z -43.514,A -90.000,B 90.000,C 0.000} C_DIS
LIN {X -103.121,Y -23.308,Z -43.422,A -90.000,B 90.000,C 0.000} C_DIS
LIN {X -102.911,Y -23.308,Z -43.181,A -90.000,B 90.000,C 0.000} C_DIS
LIN {X -102.660,Y -23.308,Z -42.905,A -90.000,B 90.000,C 0.000} C_DIS
LIN {X -102.415,Y -23.308,Z -42.699,A -90.000,B 90.000,C 0.000} C_DIS
LIN {X -102.249,Y -23.308,Z -42.581,A -90.000,B 90.000,C 0.000} C_DIS
LIN {X -102.080,Y -23.308,Z -42.456,A -90.000,B 90.000,C 0.000} C_DIS
LIN {X -101.806,Y -23.308,Z -42.279,A -90.000,B 90.000,C 0.000} C_DIS
LIN {X -101.496,Y -23.308,Z -42.113,A -90.000,B 90.000,C 0.000} C_DIS
LIN {X -101.046,Y -23.308,Z -41.919,A -90.000,B 90.000,C 0.000} C_DIS
LIN {X -100.716,Y -23.308,Z -41.799,A -90.000,B 90.000,C 0.000} C_DIS
LIN {X -100.320,Y -23.308,Z -41.715,A -90.000,B 90.000,C 0.000} C_DIS
LIN {X -99.510,Y -23.308,Z -41.588,A -90.000,B 90.000,C 0.000} C_DIS
LIN {X -99.222,Y -23.308,Z -41.550,A -90.000,B 90.000,C 0.000} C_DIS
LIN {X -98.844,Y -23.308,Z -41.521,A -90.000,B 90.000,C 0.000} C_DIS
LIN {X -98.562,Y -23.308,Z -41.518,A -90.000,B 90.000,C 0.000} C_DIS
LIN {X -98.214,Y -23.308,Z -41.518,A -90.000,B 90.000,C 0.000} C_DIS
LIN {X -97.610,Y -23.308,Z -41.532,A -90.000,B 90.000,C 0.000} C_DIS
LIN {X -97.131,Y -23.308,Z -41.562,A -90.000,B 90.000,C 0.000} C_DIS
LIN {X -96.386,Y -23.308,Z -41.636,A -90.000,B 90.000,C 0.000} C_DIS
LIN {X -96.289,Y -23.308,Z -41.649,A -90.000,B 90.000,C 0.000} C_DIS
LIN {X -96.183,Y -23.308,Z -41.494,A -90.000,B 90.000,C 0.000} C_DIS
LIN {X -95.955,Y -23.308,Z -41.111,A -90.000,B 90.000,C 0.000} C_DIS
LIN {X -95.772,Y -23.308,Z -40.827,A -90.000,B 90.000,C 0.000} C_DIS
LIN {X -95.314,Y -23.308,Z -40.281,A -90.000,B 90.000,C 0.000} C_DIS
LIN {X -95.242,Y -23.308,Z -40.169,A -90.000,B 90.000,C 0.000} C_DIS
LIN {X -95.050,Y -23.308,Z -39.963,A -90.000,B 90.000,C 0.000} C_DIS
LIN {X -94.761,Y -23.308,Z -39.671,A -90.000,B 90.000,C 0.000} C_DIS
LIN {X -94.621,Y -23.308,Z -39.490,A -90.000,B 90.000,C 0.000} C_DIS
LIN {X -94.429,Y -23.308,Z -39.284,A -90.000,B 90.000,C 0.000} C_DIS
LIN {X -94.084,Y -23.308,Z -38.978,A -90.000,B 90.000,C 0.000} C_DIS
LIN {X -93.724,Y -23.308,Z -38.608,A -90.000,B 90.000,C 0.000} C_DIS
LIN {X -93.207,Y -23.308,Z -38.179,A -90.000,B 90.000,C 0.000} C_DIS
LIN {X -92.856,Y -23.308,Z -37.940,A -90.000,B 90.000,C 0.000} C_DIS
LIN {X -92.573,Y -23.308,Z -37.702,A -90.000,B 90.000,C 0.000} C_DIS
LIN {X -92.299,Y -23.308,Z -37.537,A -90.000,B 90.000,C 0.000} C_DIS
LIN {X -92.135,Y -23.308,Z -37.445,A -90.000,B 90.000,C 0.000} C_DIS
LIN {X -91.896,Y -23.308,Z -37.270,A -90.000,B 90.000,C 0.000} C_DIS
LIN {X -91.622,Y -23.308,Z -37.105,A -90.000,B 90.000,C 0.000} C_DIS
LIN {X -91.420,Y -23.308,Z -37.005,A -90.000,B 90.000,C 0.000} C_DIS
LIN {X -90.896,Y -23.308,Z -36.699,A -90.000,B 90.000,C 0.000} C_DIS
LIN {X -90.324,Y -23.308,Z -36.422,A -90.000,B 90.000,C 0.000} C_DIS
LIN {X -90.090,Y -23.308,Z -36.290,A -90.000,B 90.000,C 0.000} C_DIS
LIN {X -89.467,Y -23.308,Z -35.954,A -90.000,B 90.000,C 0.000} C_DIS
LIN {X -89.281,Y -23.308,Z -35.858,A -90.000,B 90.000,C 0.000} C_DIS
LIN {X -89.050,Y -23.308,Z -35.722,A -90.000,B 90.000,C 0.000} C_DIS
LIN {X -88.568,Y -23.308,Z -35.463,A -90.000,B 90.000,C 0.000} C_DIS
LIN {X -88.469,Y -23.308,Z -35.399,A -90.000,B 90.000,C 0.000} C_DIS
LIN {X -88.534,Y -23.308,Z -35.216,A -90.000,B 90.000,C 0.000} C_DIS
LIN {X -88.556,Y -23.308,Z -35.086,A -90.000,B 90.000,C 0.000} C_DIS
LIN {X -88.688,Y -23.308,Z -34.864,A -90.000,B 90.000,C 0.000} C_DIS
LIN {X -88.896,Y -23.308,Z -34.266,A -90.000,B 90.000,C 0.000} C_DIS
LIN {X -88.908,Y -23.308,Z -34.060,A -90.000,B 90.000,C 0.000} C_DIS
LIN {X -88.890,Y -23.308,Z -33.977,A -90.000,B 90.000,C 0.000} C_DIS
LIN {X -88.905,Y -23.308,Z -33.404,A -90.000,B 90.000,C 0.000} C_DIS
LIN {X -88.866,Y -23.308,Z -33.229,A -90.000,B 90.000,C 0.000} C_DIS
LIN {X -88.780,Y -23.308,Z -33.071,A -90.000,B 90.000,C 0.000} C_DIS
LIN {X -88.409,Y -23.308,Z -32.667,A -90.000,B 90.000,C 0.000} C_DIS
LIN {X -88.157,Y -23.308,Z -32.342,A -90.000,B 90.000,C 0.000} C_DIS
LIN {X -88.032,Y -23.308,Z -32.214,A -90.000,B 90.000,C 0.000} C_DIS
LIN {X -87.849,Y -23.308,Z -32.103,A -90.000,B 90.000,C 0.000} C_DIS
LIN {X -87.693,Y -23.308,Z -32.015,A -90.000,B 90.000,C 0.000} C_DIS
LIN {X -87.570,Y -23.308,Z -31.971,A -90.000,B 90.000,C 0.000} C_DIS
LIN {X -86.746,Y -23.308,Z -31.633,A -90.000,B 90.000,C 0.000} C_DIS
LIN {X -86.028,Y -23.308,Z -31.205,A -90.000,B 90.000,C 0.000} C_DIS
LIN {X -85.953,Y -23.308,Z -31.101,A -90.000,B 90.000,C 0.000} C_DIS
LIN {X -85.757,Y -23.308,Z -30.751,A -90.000,B 90.000,C 0.000} C_DIS
LIN {X -85.717,Y -23.308,Z -30.641,A -90.000,B 90.000,C 0.000} C_DIS
LIN {X -85.678,Y -23.308,Z -30.475,A -90.000,B 90.000,C 0.000} C_DIS
LIN {X -85.689,Y -23.308,Z -30.285,A -90.000,B 90.000,C 0.000} C_DIS
LIN {X -85.728,Y -23.308,Z -30.104,A -90.000,B 90.000,C 0.000} C_DIS
LIN {X -85.745,Y -23.308,Z -30.069,A -90.000,B 90.000,C 0.000} C_DIS
LIN {X -85.831,Y -23.308,Z -29.889,A -90.000,B 90.000,C 0.000} C_DIS
LIN {X -85.872,Y -23.308,Z -29.787,A -90.000,B 90.000,C 0.000} C_DIS
LIN {X -85.991,Y -23.308,Z -29.573,A -90.000,B 90.000,C 0.000} C_DIS
LIN {X -86.070,Y -23.308,Z -29.349,A -90.000,B 90.000,C 0.000} C_DIS
LIN {X -86.080,Y -23.308,Z -29.272,A -90.000,B 90.000,C 0.000} C_DIS
LIN {X -86.123,Y -23.308,Z -29.082,A -90.000,B 90.000,C 0.000} C_DIS
LIN {X -86.153,Y -23.308,Z -28.847,A -90.000,B 90.000,C 0.000} C_DIS
LIN {X -86.133,Y -23.308,Z -28.610,A -90.000,B 90.000,C 0.000} C_DIS
LIN {X -86.123,Y -23.308,Z -28.538,A -90.000,B 90.000,C 0.000} C_DIS
LIN {X -86.104,Y -23.308,Z -28.454,A -90.000,B 90.000,C 0.000} C_DIS
LIN {X -85.980,Y -23.308,Z -28.037,A -90.000,B 90.000,C 0.000} C_DIS
LIN {X -85.871,Y -23.308,Z -27.776,A -90.000,B 90.000,C 0.000} C_DIS
LIN {X -85.683,Y -23.308,Z -27.425,A -90.000,B 90.000,C 0.000} C_DIS
LIN {X -85.614,Y -23.308,Z -27.311,A -90.000,B 90.000,C 0.000} C_DIS
LIN {X -85.480,Y -23.308,Z -27.103,A -90.000,B 90.000,C 0.000} C_DIS
LIN {X -84.951,Y -23.308,Z -26.368,A -90.000,B 90.000,C 0.000} C_DIS
LIN {X -84.641,Y -23.308,Z -26.013,A -90.000,B 90.000,C 0.000} C_DIS
LIN {X -84.077,Y -23.308,Z -25.432,A -90.000,B 90.000,C 0.000} C_DIS
LIN {X -83.829,Y -23.308,Z -25.192,A -90.000,B 90.000,C 0.000} C_DIS
LIN {X -83.354,Y -23.308,Z -24.739,A -90.000,B 90.000,C 0.000} C_DIS
LIN {X -82.728,Y -23.308,Z -24.155,A -90.000,B 90.000,C 0.000} C_DIS
LIN {X -82.401,Y -23.308,Z -23.880,A -90.000,B 90.000,C 0.000} C_DIS
LIN {X -81.950,Y -23.308,Z -23.525,A -90.000,B 90.000,C 0.000} C_DIS
LIN {X -81.647,Y -23.308,Z -23.319,A -90.000,B 90.000,C 0.000} C_DIS
LIN {X -81.373,Y -23.308,Z -23.154,A -90.000,B 90.000,C 0.000} C_DIS
LIN {X -80.974,Y -23.308,Z -22.947,A -90.000,B 90.000,C 0.000} C_DIS
LIN {X -80.622,Y -23.308,Z -22.779,A -90.000,B 90.000,C 0.000} C_DIS
LIN {X -80.423,Y -23.308,Z -22.699,A -90.000,B 90.000,C 0.000} C_DIS
LIN {X -80.334,Y -23.308,Z -22.672,A -90.000,B 90.000,C 0.000} C_DIS
LIN {X -79.876,Y -23.308,Z -22.566,A -90.000,B 90.000,C 0.000} C_DIS
LIN {X -79.596,Y -23.308,Z -22.534,A -90.000,B 90.000,C 0.000} C_DIS
LIN {X -79.112,Y -23.308,Z -22.567,A -90.000,B 90.000,C 0.000} C_DIS
LIN {X -78.843,Y -23.308,Z -22.586,A -90.000,B 90.000,C 0.000} C_DIS
LIN {X -78.755,Y -23.308,Z -22.600,A -90.000,B 90.000,C 0.000} C_DIS
LIN {X -78.473,Y -23.308,Z -22.670,A -90.000,B 90.000,C 0.000} C_DIS
LIN {X -78.216,Y -23.308,Z -22.784,A -90.000,B 90.000,C 0.000} C_DIS
LIN {X -77.643,Y -23.308,Z -23.175,A -90.000,B 90.000,C 0.000} C_DIS
LIN {X -77.524,Y -23.308,Z -23.261,A -90.000,B 90.000,C 0.000} C_DIS
LIN {X -77.323,Y -23.308,Z -23.457,A -90.000,B 90.000,C 0.000} C_DIS
LIN {X -76.918,Y -23.308,Z -23.954,A -90.000,B 90.000,C 0.000} C_DIS
LIN {X -76.526,Y -23.308,Z -24.456,A -90.000,B 90.000,C 0.000} C_DIS
LIN {X -76.172,Y -23.308,Z -24.794,A -90.000,B 90.000,C 0.000} C_DIS
LIN {X -75.699,Y -23.308,Z -25.074,A -90.000,B 90.000,C 0.000} C_DIS
LIN {X -75.508,Y -23.308,Z -25.178,A -90.000,B 90.000,C 0.000} C_DIS
LIN {X -74.840,Y -23.308,Z -25.618,A -90.000,B 90.000,C 0.000} C_DIS
LIN {X -74.606,Y -23.308,Z -25.777,A -90.000,B 90.000,C 0.000} C_DIS
LIN {X -74.385,Y -23.308,Z -25.935,A -90.000,B 90.000,C 0.000} C_DIS
LIN {X -74.376,Y -23.308,Z -25.943,A -90.000,B 90.000,C 0.000} C_DIS
LIN {X -74.191,Y -23.308,Z -26.123,A -90.000,B 90.000,C 0.000} C_DIS
LIN {X -73.391,Y -23.308,Z -26.946,A -90.000,B 90.000,C 0.000} C_DIS
LIN {X -73.227,Y -23.308,Z -27.176,A -90.000,B 90.000,C 0.000} C_DIS
LIN {X -73.100,Y -23.308,Z -27.444,A -90.000,B 90.000,C 0.000} C_DIS
LIN {X -72.834,Y -23.308,Z -28.029,A -90.000,B 90.000,C 0.000} C_DIS
LIN {X -72.694,Y -23.308,Z -28.292,A -90.000,B 90.000,C 0.000} C_DIS
LIN {X -72.574,Y -23.308,Z -28.546,A -90.000,B 90.000,C 0.000} C_DIS
LIN {X -72.500,Y -23.308,Z -28.819,A -90.000,B 90.000,C 0.000} C_DIS
LIN {X -72.444,Y -23.308,Z -29.081,A -90.000,B 90.000,C 0.000} C_DIS
LIN {X -72.414,Y -23.308,Z -29.369,A -90.000,B 90.000,C 0.000} C_DIS
LIN {X -72.389,Y -23.308,Z -29.688,A -90.000,B 90.000,C 0.000} C_DIS
LIN {X -72.358,Y -23.308,Z -30.209,A -90.000,B 90.000,C 0.000} C_DIS
LIN {X -72.360,Y -23.308,Z -30.623,A -90.000,B 90.000,C 0.000} C_DIS
LIN {X -72.433,Y -23.308,Z -32.079,A -90.000,B 90.000,C 0.000} C_DIS
LIN {X -72.481,Y -23.308,Z -32.356,A -90.000,B 90.000,C 0.000} C_DIS
LIN {X -72.493,Y -23.308,Z -32.401,A -90.000,B 90.000,C 0.000} C_DIS
LIN {X -72.540,Y -23.308,Z -33.072,A -90.000,B 90.000,C 0.000} C_DIS
LIN {X -72.510,Y -23.308,Z -33.708,A -90.000,B 90.000,C 0.000} C_DIS
LIN {X -72.206,Y -23.308,Z -34.538,A -90.000,B 90.000,C 0.000} C_DIS
LIN {X -71.500,Y -23.308,Z -35.187,A -90.000,B 90.000,C 0.000} C_DIS
LIN {X -70.648,Y -23.308,Z -35.686,A -90.000,B 90.000,C 0.000} C_DIS
LIN {X -70.481,Y -23.308,Z -35.775,A -90.000,B 90.000,C 0.000} C_DIS
LIN {X -69.898,Y -23.308,Z -36.028,A -90.000,B 90.000,C 0.000} C_DIS
LIN {X -68.699,Y -23.308,Z -36.619,A -90.000,B 90.000,C 0.000} C_DIS
LIN {X -67.629,Y -23.308,Z -37.195,A -90.000,B 90.000,C 0.000} C_DIS
LIN {X -65.714,Y -23.308,Z -38.141,A -90.000,B 90.000,C 0.000} C_DIS
LIN {X -65.181,Y -23.308,Z -38.426,A -90.000,B 90.000,C 0.000} C_DIS
LIN {X -62.919,Y -23.308,Z -39.489,A -90.000,B 90.000,C 0.000} C_DIS
LIN {X -62.598,Y -23.308,Z -39.647,A -90.000,B 90.000,C 0.000} C_DIS
LIN {X -60.269,Y -23.308,Z -40.655,A -90.000,B 90.000,C 0.000} C_DIS
LIN {X -59.935,Y -23.308,Z -40.801,A -90.000,B 90.000,C 0.000} C_DIS
LIN {X -57.382,Y -23.308,Z -41.772,A -90.000,B 90.000,C 0.000} C_DIS
LIN {X -56.570,Y -23.308,Z -42.038,A -90.000,B 90.000,C 0.000} C_DIS
LIN {X -54.608,Y -23.308,Z -42.693,A -90.000,B 90.000,C 0.000} C_DIS
LIN {X -54.126,Y -23.308,Z -42.843,A -90.000,B 90.000,C 0.000} C_DIS
LIN {X -51.780,Y -23.308,Z -43.526,A -90.000,B 90.000,C 0.000} C_DIS
LIN {X -49.990,Y -23.308,Z -44.009,A -90.000,B 90.000,C 0.000} C_DIS
LIN {X -48.950,Y -23.308,Z -44.274,A -90.000,B 90.000,C 0.000} C_DIS
LIN {X -48.395,Y -23.308,Z -44.397,A -90.000,B 90.000,C 0.000} C_DIS
LIN {X -47.429,Y -23.308,Z -44.629,A -90.000,B 90.000,C 0.000} C_DIS
LIN {X -46.358,Y -23.308,Z -44.865,A -90.000,B 90.000,C 0.000} C_DIS
LIN {X -45.970,Y -23.308,Z -44.966,A -90.000,B 90.000,C 0.000} C_DIS
LIN {X -44.685,Y -23.308,Z -45.232,A -90.000,B 90.000,C 0.000} C_DIS
LIN {X -44.364,Y -23.308,Z -45.304,A -90.000,B 90.000,C 0.000} C_DIS
LIN {X -42.865,Y -23.308,Z -45.679,A -90.000,B 90.000,C 0.000} C_DIS
LIN {X -42.368,Y -23.308,Z -45.788,A -90.000,B 90.000,C 0.000} C_DIS
LIN {X -39.562,Y -23.308,Z -46.514,A -90.000,B 90.000,C 0.000} C_DIS
LIN {X -39.214,Y -23.308,Z -46.621,A -90.000,B 90.000,C 0.000} C_DIS
LIN {X -36.467,Y -23.308,Z -47.422,A -90.000,B 90.000,C 0.000} C_DIS
LIN {X -35.904,Y -23.308,Z -47.609,A -90.000,B 90.000,C 0.000} C_DIS
LIN {X -34.479,Y -23.308,Z -48.087,A -90.000,B 90.000,C 0.000} C_DIS
LIN {X -33.005,Y -23.308,Z -48.552,A -90.000,B 90.000,C 0.000} C_DIS
LIN {X -31.582,Y -23.308,Z -49.040,A -90.000,B 90.000,C 0.000} C_DIS
LIN {X -32.098,Y -23.308,Z -48.505,A -90.000,B 90.000,C 0.000} C_DIS
LIN {X -32.151,Y -23.308,Z -48.439,A -90.000,B 90.000,C 0.000} C_DIS
LIN {X -32.249,Y -23.308,Z -48.299,A -90.000,B 90.000,C 0.000} C_DIS
LIN {X -32.284,Y -23.308,Z -48.206,A -90.000,B 90.000,C 0.000} C_DIS
LIN {X -32.340,Y -23.308,Z -48.049,A -90.000,B 90.000,C 0.000} C_DIS
LIN {X -32.798,Y -23.308,Z -46.677,A -90.000,B 90.000,C 0.000} C_DIS
LIN {X -32.809,Y -23.308,Z -46.498,A -90.000,B 90.000,C 0.000} C_DIS
LIN {X -32.807,Y -23.308,Z -46.220,A -90.000,B 90.000,C 0.000} C_DIS
LIN {X -32.764,Y -23.308,Z -46.010,A -90.000,B 90.000,C 0.000} C_DIS
LIN {X -32.683,Y -23.308,Z -45.887,A -90.000,B 90.000,C 0.000} C_DIS
LIN {X -32.557,Y -23.308,Z -45.759,A -90.000,B 90.000,C 0.000} C_DIS
LIN {X -31.924,Y -23.308,Z -45.285,A -90.000,B 90.000,C 0.000} C_DIS
LIN {X -30.935,Y -23.308,Z -44.683,A -90.000,B 90.000,C 0.000} C_DIS
LIN {X -30.779,Y -23.308,Z -44.595,A -90.000,B 90.000,C 0.000} C_DIS
LIN {X -30.605,Y -23.308,Z -44.552,A -90.000,B 90.000,C 0.000} C_DIS
LIN {X -29.168,Y -23.308,Z -44.572,A -90.000,B 90.000,C 0.000} C_DIS
LIN {X -28.756,Y -23.308,Z -44.582,A -90.000,B 90.000,C 0.000} C_DIS
LIN {X -28.253,Y -23.308,Z -44.569,A -90.000,B 90.000,C 0.000} C_DIS
LIN {X -27.058,Y -23.308,Z -44.548,A -90.000,B 90.000,C 0.000} C_DIS
LIN {X -26.379,Y -23.308,Z -44.575,A -90.000,B 90.000,C 0.000} C_DIS
LIN {X -25.775,Y -23.308,Z -44.493,A -90.000,B 90.000,C 0.000} C_DIS
LIN {X -24.823,Y -23.308,Z -44.419,A -90.000,B 90.000,C 0.000} C_DIS
LIN {X -24.586,Y -23.308,Z -44.416,A -90.000,B 90.000,C 0.000} C_DIS
LIN {X -24.257,Y -23.308,Z -44.425,A -90.000,B 90.000,C 0.000} C_DIS
LIN {X -23.932,Y -23.308,Z -44.391,A -90.000,B 90.000,C 0.000} C_DIS
LIN {X -22.199,Y -23.308,Z -44.305,A -90.000,B 90.000,C 0.000} C_DIS
LIN {X -20.288,Y -23.308,Z -44.012,A -90.000,B 90.000,C 0.000} C_DIS
LIN {X -19.879,Y -23.308,Z -43.999,A -90.000,B 90.000,C 0.000} C_DIS
LIN {X -19.381,Y -23.308,Z -43.974,A -90.000,B 90.000,C 0.000} C_DIS
LIN {X -17.259,Y -23.308,Z -43.902,A -90.000,B 90.000,C 0.000} C_DIS
LIN {X -16.358,Y -23.308,Z -43.894,A -90.000,B 90.000,C 0.000} C_DIS
LIN {X -15.132,Y -23.308,Z -43.877,A -90.000,B 90.000,C 0.000} C_DIS
LIN {X -14.843,Y -23.308,Z -43.874,A -90.000,B 90.000,C 0.000} C_DIS
LIN {X -14.124,Y -23.308,Z -43.883,A -90.000,B 90.000,C 0.000} C_DIS
LIN {X -13.062,Y -23.308,Z -43.957,A -90.000,B 90.000,C 0.000} C_DIS
LIN {X -11.534,Y -23.308,Z -44.134,A -90.000,B 90.000,C 0.000} C_DIS
LIN {X -10.791,Y -23.308,Z -44.223,A -90.000,B 90.000,C 0.000} C_DIS
LIN {X -9.347,Y -23.308,Z -44.456,A -90.000,B 90.000,C 0.000} C_DIS
LIN {X -7.553,Y -23.308,Z -44.781,A -90.000,B 90.000,C 0.000} C_DIS
LIN {X -7.147,Y -23.308,Z -44.873,A -90.000,B 90.000,C 0.000} C_DIS
LIN {X -6.909,Y -23.308,Z -44.932,A -90.000,B 90.000,C 0.000} C_DIS
LIN {X -5.771,Y -23.308,Z -45.229,A -90.000,B 90.000,C 0.000} C_DIS
LIN {X -4.419,Y -23.308,Z -45.591,A -90.000,B 90.000,C 0.000} C_DIS
LIN {X -2.421,Y -23.308,Z -46.341,A -90.000,B 90.000,C 0.000} C_DIS
LIN {X -2.315,Y -23.308,Z -46.374,A -90.000,B 90.000,C 0.000} C_DIS
LIN {X -2.019,Y -23.308,Z -46.495,A -90.000,B 90.000,C 0.000} C_DIS
LIN {X -1.832,Y -23.308,Z -46.578,A -90.000,B 90.000,C 0.000} C_DIS
LIN {X -1.137,Y -23.308,Z -46.901,A -90.000,B 90.000,C 0.000} C_DIS
LIN {X -0.376,Y -23.308,Z -47.188,A -90.000,B 90.000,C 0.000} C_DIS
LIN {X -0.094,Y -23.308,Z -47.306,A -90.000,B 90.000,C 0.000} C_DIS
LIN {X 0.146,Y -23.308,Z -47.423,A -90.000,B 90.000,C 0.000} C_DIS
LIN {X 1.357,Y -23.308,Z -47.906,A -90.000,B 90.000,C 0.000} C_DIS
LIN {X 2.457,Y -23.308,Z -48.330,A -90.000,B 90.000,C 0.000} C_DIS
LIN {X 2.727,Y -23.308,Z -48.415,A -90.000,B 90.000,C 0.000} C_DIS
LIN {X 3.361,Y -23.308,Z -48.593,A -90.000,B 90.000,C 0.000} C_DIS
LIN {X 4.229,Y -23.308,Z -48.882,A -90.000,B 90.000,C 0.000} C_DIS
LIN {X 5.297,Y -23.308,Z -49.162,A -90.000,B 90.000,C 0.000} C_DIS
LIN {X 5.774,Y -23.308,Z -49.309,A -90.000,B 90.000,C 0.000} C_DIS
LIN {X 6.678,Y -23.308,Z -49.539,A -90.000,B 90.000,C 0.000} C_DIS
LIN {X 7.362,Y -23.308,Z -49.742,A -90.000,B 90.000,C 0.000} C_DIS
LIN {X 8.303,Y -23.308,Z -49.981,A -90.000,B 90.000,C 0.000} C_DIS
LIN {X 8.641,Y -23.308,Z -50.074,A -90.000,B 90.000,C 0.000} C_DIS
LIN {X 9.297,Y -23.308,Z -50.276,A -90.000,B 90.000,C 0.000} C_DIS
LIN {X 10.156,Y -23.308,Z -50.507,A -90.000,B 90.000,C 0.000} C_DIS
LIN {X 10.221,Y -23.308,Z -50.527,A -90.000,B 90.000,C 0.000} C_DIS
LIN {X 11.441,Y -23.308,Z -50.870,A -90.000,B 90.000,C 0.000} C_DIS
LIN {X 11.762,Y -23.308,Z -50.520,A -90.000,B 90.000,C 0.000} C_DIS
LIN {X 11.819,Y -23.308,Z -50.468,A -90.000,B 90.000,C 0.000} C_DIS
LIN {X 12.137,Y -23.308,Z -49.972,A -90.000,B 90.000,C 0.000} C_DIS
LIN {X 12.448,Y -23.308,Z -49.477,A -90.000,B 90.000,C 0.000} C_DIS
LIN {X 12.549,Y -23.308,Z -49.320,A -90.000,B 90.000,C 0.000} C_DIS
LIN {X 12.740,Y -23.308,Z -49.116,A -90.000,B 90.000,C 0.000} C_DIS
LIN {X 12.752,Y -23.308,Z -49.106,A -90.000,B 90.000,C 0.000} C_DIS
LIN {X 12.965,Y -23.308,Z -48.946,A -90.000,B 90.000,C 0.000} C_DIS
LIN {X 13.131,Y -23.308,Z -48.826,A -90.000,B 90.000,C 0.000} C_DIS
LIN {X 13.213,Y -23.308,Z -48.725,A -90.000,B 90.000,C 0.000} C_DIS
LIN {X 13.400,Y -23.308,Z -48.524,A -90.000,B 90.000,C 0.000} C_DIS
LIN {X 13.626,Y -23.308,Z -48.355,A -90.000,B 90.000,C 0.000} C_DIS
LIN {X 14.246,Y -23.308,Z -47.941,A -90.000,B 90.000,C 0.000} C_DIS
LIN {X 14.523,Y -23.308,Z -47.722,A -90.000,B 90.000,C 0.000} C_DIS
LIN {X 14.793,Y -23.308,Z -47.560,A -90.000,B 90.000,C 0.000} C_DIS
LIN {X 14.964,Y -23.308,Z -47.472,A -90.000,B 90.000,C 0.000} C_DIS
LIN {X 15.310,Y -23.308,Z -47.251,A -90.000,B 90.000,C 0.000} C_DIS
LIN {X 15.611,Y -23.308,Z -47.069,A -90.000,B 90.000,C 0.000} C_DIS
LIN {X 15.907,Y -23.308,Z -46.949,A -90.000,B 90.000,C 0.000} C_DIS
LIN {X 16.783,Y -23.308,Z -46.648,A -90.000,B 90.000,C 0.000} C_DIS
LIN {X 16.939,Y -23.308,Z -46.591,A -90.000,B 90.000,C 0.000} C_DIS
LIN {X 17.156,Y -23.308,Z -46.490,A -90.000,B 90.000,C 0.000} C_DIS
LIN {X 17.486,Y -23.308,Z -46.370,A -90.000,B 90.000,C 0.000} C_DIS
LIN {X 18.022,Y -23.308,Z -46.215,A -90.000,B 90.000,C 0.000} C_DIS
LIN {X 18.258,Y -23.308,Z -46.152,A -90.000,B 90.000,C 0.000} C_DIS
LIN {X 18.635,Y -23.308,Z -46.041,A -90.000,B 90.000,C 0.000} C_DIS
LIN {X 19.188,Y -23.308,Z -45.898,A -90.000,B 90.000,C 0.000} C_DIS
LIN {X 19.555,Y -23.308,Z -45.820,A -90.000,B 90.000,C 0.000} C_DIS
LIN {X 19.666,Y -23.308,Z -45.802,A -90.000,B 90.000,C 0.000} C_DIS
LIN {X 20.383,Y -23.308,Z -45.616,A -90.000,B 90.000,C 0.000} C_DIS
LIN {X 20.886,Y -23.308,Z -45.492,A -90.000,B 90.000,C 0.000} C_DIS
LIN {X 21.266,Y -23.308,Z -45.405,A -90.000,B 90.000,C 0.000} C_DIS
LIN {X 21.977,Y -23.308,Z -45.293,A -90.000,B 90.000,C 0.000} C_DIS
LIN {X 22.892,Y -23.308,Z -45.051,A -90.000,B 90.000,C 0.000} C_DIS
LIN {X 23.933,Y -23.308,Z -44.870,A -90.000,B 90.000,C 0.000} C_DIS
LIN {X 24.372,Y -23.308,Z -44.748,A -90.000,B 90.000,C 0.000} C_DIS
LIN {X 25.133,Y -23.308,Z -44.606,A -90.000,B 90.000,C 0.000} C_DIS
LIN {X 25.461,Y -23.308,Z -44.534,A -90.000,B 90.000,C 0.000} C_DIS
LIN {X 25.909,Y -23.308,Z -44.450,A -90.000,B 90.000,C 0.000} C_DIS
LIN {X 25.974,Y -23.308,Z -44.440,A -90.000,B 90.000,C 0.000} C_DIS
LIN {X 26.148,Y -23.308,Z -44.397,A -90.000,B 90.000,C 0.000} C_DIS
LIN {X 26.225,Y -23.308,Z -44.383,A -90.000,B 90.000,C 0.000} C_DIS
LIN {X 26.509,Y -23.308,Z -44.316,A -90.000,B 90.000,C 0.000} C_DIS
LIN {X 27.162,Y -23.308,Z -44.174,A -90.000,B 90.000,C 0.000} C_DIS
LIN {X 27.749,Y -23.308,Z -44.070,A -90.000,B 90.000,C 0.000} C_DIS
LIN {X 28.029,Y -23.308,Z -44.010,A -90.000,B 90.000,C 0.000} C_DIS
LIN {X 28.624,Y -23.308,Z -43.856,A -90.000,B 90.000,C 0.000} C_DIS
LIN {X 29.122,Y -23.308,Z -43.736,A -90.000,B 90.000,C 0.000} C_DIS
LIN {X 29.705,Y -23.308,Z -43.568,A -90.000,B 90.000,C 0.000} C_DIS
LIN {X 30.222,Y -23.308,Z -43.415,A -90.000,B 90.000,C 0.000} C_DIS
LIN {X 30.610,Y -23.308,Z -43.290,A -90.000,B 90.000,C 0.000} C_DIS
LIN {X 32.343,Y -23.308,Z -42.684,A -90.000,B 90.000,C 0.000} C_DIS
LIN {X 33.285,Y -23.308,Z -42.357,A -90.000,B 90.000,C 0.000} C_DIS
LIN {X 34.611,Y -23.308,Z -41.882,A -90.000,B 90.000,C 0.000} C_DIS
LIN {X 35.365,Y -23.308,Z -41.640,A -90.000,B 90.000,C 0.000} C_DIS
LIN {X 35.776,Y -23.308,Z -41.513,A -90.000,B 90.000,C 0.000} C_DIS
LIN {X 36.853,Y -23.308,Z -41.212,A -90.000,B 90.000,C 0.000} C_DIS
LIN {X 37.137,Y -23.308,Z -41.130,A -90.000,B 90.000,C 0.000} C_DIS
LIN {X 38.288,Y -23.308,Z -40.865,A -90.000,B 90.000,C 0.000} C_DIS
LIN {X 39.062,Y -23.308,Z -40.706,A -90.000,B 90.000,C 0.000} C_DIS
LIN {X 40.552,Y -23.308,Z -40.512,A -90.000,B 90.000,C 0.000} C_DIS
LIN {X 40.947,Y -23.308,Z -40.465,A -90.000,B 90.000,C 0.000} C_DIS
LIN {X 41.461,Y -23.308,Z -40.427,A -90.000,B 90.000,C 0.000} C_DIS
LIN {X 42.240,Y -23.308,Z -40.403,A -90.000,B 90.000,C 0.000} C_DIS
LIN {X 42.930,Y -23.308,Z -40.400,A -90.000,B 90.000,C 0.000} C_DIS
LIN {X 43.445,Y -23.308,Z -40.411,A -90.000,B 90.000,C 0.000} C_DIS
LIN {X 43.920,Y -23.308,Z -40.434,A -90.000,B 90.000,C 0.000} C_DIS
LIN {X 44.199,Y -23.308,Z -40.457,A -90.000,B 90.000,C 0.000} C_DIS
LIN {X 45.363,Y -23.308,Z -40.618,A -90.000,B 90.000,C 0.000} C_DIS
LIN {X 45.833,Y -23.308,Z -40.691,A -90.000,B 90.000,C 0.000} C_DIS
LIN {X 47.136,Y -23.308,Z -40.978,A -90.000,B 90.000,C 0.000} C_DIS
LIN {X 47.698,Y -23.308,Z -41.109,A -90.000,B 90.000,C 0.000} C_DIS
LIN {X 47.894,Y -23.308,Z -41.161,A -90.000,B 90.000,C 0.000} C_DIS
LIN {X 48.161,Y -23.308,Z -41.236,A -90.000,B 90.000,C 0.000} C_DIS
LIN {X 48.572,Y -23.308,Z -41.382,A -90.000,B 90.000,C 0.000} C_DIS
LIN {X 50.353,Y -23.308,Z -42.089,A -90.000,B 90.000,C 0.000} C_DIS
LIN {X 51.462,Y -23.308,Z -42.572,A -90.000,B 90.000,C 0.000} C_DIS
LIN {X 51.890,Y -23.308,Z -42.797,A -90.000,B 90.000,C 0.000} C_DIS
LIN {X 52.462,Y -23.308,Z -43.102,A -90.000,B 90.000,C 0.000} C_DIS
LIN {X 53.467,Y -23.308,Z -43.660,A -90.000,B 90.000,C 0.000} C_DIS
LIN {X 54.560,Y -23.308,Z -44.273,A -90.000,B 90.000,C 0.000} C_DIS
LIN {X 54.979,Y -23.308,Z -44.558,A -90.000,B 90.000,C 0.000} C_DIS
LIN {X 56.590,Y -23.308,Z -45.722,A -90.000,B 90.000,C 0.000} C_DIS
LIN {X 57.355,Y -23.308,Z -46.264,A -90.000,B 90.000,C 0.000} C_DIS
LIN {X 57.728,Y -23.308,Z -46.577,A -90.000,B 90.000,C 0.000} C_DIS
LIN {X 59.270,Y -23.308,Z -47.895,A -90.000,B 90.000,C 0.000} C_DIS
LIN {X 59.847,Y -23.308,Z -48.393,A -90.000,B 90.000,C 0.000} C_DIS
LIN {X 61.050,Y -23.308,Z -49.523,A -90.000,B 90.000,C 0.000} C_DIS
LIN {X 61.774,Y -23.308,Z -50.212,A -90.000,B 90.000,C 0.000} C_DIS
LIN {X 62.069,Y -23.308,Z -50.480,A -90.000,B 90.000,C 0.000} C_DIS
LIN {X 63.583,Y -23.308,Z -51.911,A -90.000,B 90.000,C 0.000} C_DIS
LIN {X 64.298,Y -23.308,Z -52.499,A -90.000,B 90.000,C 0.000} C_DIS
LIN {X 65.129,Y -23.308,Z -53.190,A -90.000,B 90.000,C 0.000} C_DIS
LIN {X 65.207,Y -23.308,Z -53.257,A -90.000,B 90.000,C 0.000} C_DIS
LIN {X 65.473,Y -23.308,Z -53.444,A -90.000,B 90.000,C 0.000} C_DIS
LIN {X 66.886,Y -23.308,Z -54.389,A -90.000,B 90.000,C 0.000} C_DIS
LIN {X 68.896,Y -23.308,Z -55.620,A -90.000,B 90.000,C 0.000} C_DIS
LIN {X 68.999,Y -23.308,Z -55.682,A -90.000,B 90.000,C 0.000} C_DIS
LIN {X 71.100,Y -23.308,Z -56.973,A -90.000,B 90.000,C 0.000} C_DIS
LIN {X 71.537,Y -23.308,Z -57.265,A -90.000,B 90.000,C 0.000} C_DIS
LIN {X 73.141,Y -23.308,Z -58.364,A -90.000,B 90.000,C 0.000} C_DIS
LIN {X 73.353,Y -23.308,Z -58.507,A -90.000,B 90.000,C 0.000} C_DIS
LIN {X 73.434,Y -23.308,Z -58.569,A -90.000,B 90.000,C 0.000} C_DIS
LIN {X 73.724,Y -23.308,Z -58.806,A -90.000,B 90.000,C 0.000} C_DIS
LIN {X 74.287,Y -23.308,Z -59.276,A -90.000,B 90.000,C 0.000} C_DIS
LIN {X 75.340,Y -23.308,Z -60.191,A -90.000,B 90.000,C 0.000} C_DIS
LIN {X 75.677,Y -23.308,Z -60.527,A -90.000,B 90.000,C 0.000} C_DIS
LIN {X 75.964,Y -23.308,Z -60.818,A -90.000,B 90.000,C 0.000} C_DIS
LIN {X 77.015,Y -23.308,Z -61.943,A -90.000,B 90.000,C 0.000} C_DIS
LIN {X 77.351,Y -23.308,Z -62.354,A -90.000,B 90.000,C 0.000} C_DIS
LIN {X 78.292,Y -23.308,Z -63.550,A -90.000,B 90.000,C 0.000} C_DIS
LIN {X 78.535,Y -23.308,Z -63.873,A -90.000,B 90.000,C 0.000} C_DIS
LIN {X 78.593,Y -23.308,Z -63.951,A -90.000,B 90.000,C 0.000} C_DIS
LIN {X 78.846,Y -23.308,Z -64.316,A -90.000,B 90.000,C 0.000} C_DIS
LIN {X 79.034,Y -23.308,Z -63.681,A -90.000,B 90.000,C 0.000} C_DIS
LIN {X 79.745,Y -23.308,Z -61.550,A -90.000,B 90.000,C 0.000} C_DIS
LIN {X 79.783,Y -23.308,Z -61.448,A -90.000,B 90.000,C 0.000} C_DIS
LIN {X 80.307,Y -23.308,Z -59.771,A -90.000,B 90.000,C 0.000} C_DIS
LIN {X 80.465,Y -23.308,Z -59.303,A -90.000,B 90.000,C 0.000} C_DIS
LIN {X 81.203,Y -23.308,Z -57.299,A -90.000,B 90.000,C 0.000} C_DIS
LIN {X 81.700,Y -23.308,Z -56.182,A -90.000,B 90.000,C 0.000} C_DIS
LIN {X 82.136,Y -23.308,Z -55.104,A -90.000,B 90.000,C 0.000} C_DIS
LIN {X 82.335,Y -23.308,Z -54.666,A -90.000,B 90.000,C 0.000} C_DIS
LIN {X 83.349,Y -23.308,Z -52.780,A -90.000,B 90.000,C 0.000} C_DIS
LIN {X 83.577,Y -23.308,Z -52.389,A -90.000,B 90.000,C 0.000} C_DIS
LIN {X 84.742,Y -23.308,Z -50.678,A -90.000,B 90.000,C 0.000} C_DIS
LIN {X 85.025,Y -23.308,Z -50.291,A -90.000,B 90.000,C 0.000} C_DIS
LIN {X 86.337,Y -23.308,Z -48.714,A -90.000,B 90.000,C 0.000} C_DIS
LIN {X 86.664,Y -23.308,Z -48.352,A -90.000,B 90.000,C 0.000} C_DIS
LIN {X 88.117,Y -23.308,Z -46.880,A -90.000,B 90.000,C 0.000} C_DIS
LIN {X 88.517,Y -23.308,Z -46.520,A -90.000,B 90.000,C 0.000} C_DIS
LIN {X 90.061,Y -23.308,Z -45.164,A -90.000,B 90.000,C 0.000} C_DIS
LIN {X 91.729,Y -23.308,Z -43.867,A -90.000,B 90.000,C 0.000} C_DIS
LIN {X 92.110,Y -23.308,Z -43.588,A -90.000,B 90.000,C 0.000} C_DIS
LIN {X 93.780,Y -23.308,Z -42.419,A -90.000,B 90.000,C 0.000} C_DIS
LIN {X 95.435,Y -23.308,Z -41.372,A -90.000,B 90.000,C 0.000} C_DIS
LIN {X 95.906,Y -23.308,Z -41.097,A -90.000,B 90.000,C 0.000} C_DIS
LIN {X 97.376,Y -23.308,Z -40.260,A -90.000,B 90.000,C 0.000} C_DIS
LIN {X 97.447,Y -23.308,Z -40.223,A -90.000,B 90.000,C 0.000} C_DIS
LIN {X 98.805,Y -23.308,Z -39.523,A -90.000,B 90.000,C 0.000} C_DIS
LIN {X 100.266,Y -23.308,Z -38.830,A -90.000,B 90.000,C 0.000} C_DIS
LIN {X 102.116,Y -23.308,Z -37.992,A -90.000,B 90.000,C 0.000} C_DIS
LIN {X 103.603,Y -23.308,Z -37.329,A -90.000,B 90.000,C 0.000} C_DIS
LIN {X 104.541,Y -23.308,Z -36.915,A -90.000,B 90.000,C 0.000} C_DIS
LIN {X 105.369,Y -23.308,Z -36.566,A -90.000,B 90.000,C 0.000} C_DIS
LIN {X 106.885,Y -23.308,Z -35.963,A -90.000,B 90.000,C 0.000} C_DIS
LIN {X 107.409,Y -23.308,Z -35.765,A -90.000,B 90.000,C 0.000} C_DIS
LIN {X 107.855,Y -23.308,Z -35.604,A -90.000,B 90.000,C 0.000} C_DIS
LIN {X 108.317,Y -23.308,Z -35.448,A -90.000,B 90.000,C 0.000} C_DIS
LIN {X 108.745,Y -23.308,Z -35.333,A -90.000,B 90.000,C 0.000} C_DIS
LIN {X 109.221,Y -23.308,Z -35.225,A -90.000,B 90.000,C 0.000} C_DIS
LIN {X 109.663,Y -23.308,Z -35.167,A -90.000,B 90.000,C 0.000} C_DIS
LIN {X 110.108,Y -23.308,Z -35.113,A -90.000,B 90.000,C 0.000} C_DIS
LIN {X 110.596,Y -23.308,Z -35.105,A -90.000,B 90.000,C 0.000} C_DIS
LIN {X 110.949,Y -23.308,Z -35.117,A -90.000,B 90.000,C 0.000} C_DIS
LIN {X 111.447,Y -23.308,Z -35.160,A -90.000,B 90.000,C 0.000} C_DIS
LIN {X 112.068,Y -23.308,Z -35.277,A -90.000,B 90.000,C 0.000} C_DIS
LIN {X 112.405,Y -23.308,Z -35.362,A -90.000,B 90.000,C 0.000} C_DIS
LIN {X 112.935,Y -23.308,Z -35.522,A -90.000,B 90.000,C 0.000} C_DIS
LIN {X 113.055,Y -23.308,Z -35.560,A -90.000,B 90.000,C 0.000} C_DIS
LIN {X 113.505,Y -23.308,Z -35.746,A -90.000,B 90.000,C 0.000} C_DIS
LIN {X 113.979,Y -23.308,Z -35.973,A -90.000,B 90.000,C 0.000} C_DIS
LIN {X 114.420,Y -23.308,Z -36.211,A -90.000,B 90.000,C 0.000} C_DIS
LIN {X 114.540,Y -23.308,Z -36.286,A -90.000,B 90.000,C 0.000} C_DIS
LIN {X 114.953,Y -23.308,Z -36.567,A -90.000,B 90.000,C 0.000} C_DIS
LIN {X 115.050,Y -23.308,Z -36.644,A -90.000,B 90.000,C 0.000} C_DIS
LIN {X 115.431,Y -23.308,Z -36.965,A -90.000,B 90.000,C 0.000} C_DIS
LIN {X 115.513,Y -23.308,Z -37.039,A -90.000,B 90.000,C 0.000} C_DIS
LIN {X 115.636,Y -23.308,Z -37.166,A -90.000,B 90.000,C 0.000} C_DIS
LIN {X 115.933,Y -23.308,Z -37.475,A -90.000,B 90.000,C 0.000} C_DIS
LIN {X 116.081,Y -23.308,Z -37.633,A -90.000,B 90.000,C 0.000} C_DIS
LIN {X 116.439,Y -23.308,Z -38.088,A -90.000,B 90.000,C 0.000} C_DIS
LIN {X 116.700,Y -23.308,Z -38.500,A -90.000,B 90.000,C 0.000} C_DIS
LIN {X 116.930,Y -23.308,Z -38.965,A -90.000,B 90.000,C 0.000} C_DIS
LIN {X 117.059,Y -23.308,Z -39.250,A -90.000,B 90.000,C 0.000} C_DIS
LIN {X 117.105,Y -23.308,Z -39.366,A -90.000,B 90.000,C 0.000} C_DIS
LIN {X 117.260,Y -23.308,Z -39.781,A -90.000,B 90.000,C 0.000} C_DIS
LIN {X 117.391,Y -23.308,Z -40.284,A -90.000,B 90.000,C 0.000} C_DIS
LIN {X 117.462,Y -23.308,Z -40.593,A -90.000,B 90.000,C 0.000} C_DIS
LIN {X 117.541,Y -23.308,Z -41.113,A -90.000,B 90.000,C 0.000} C_DIS
LIN {X 117.596,Y -23.308,Z -41.528,A -90.000,B 90.000,C 0.000} C_DIS
LIN {X 117.630,Y -23.308,Z -41.874,A -90.000,B 90.000,C 0.000} C_DIS
LIN {X 117.660,Y -23.308,Z -42.479,A -90.000,B 90.000,C 0.000} C_DIS
LIN {X 117.668,Y -23.308,Z -42.699,A -90.000,B 90.000,C 0.000} C_DIS
LIN {X 117.664,Y -23.308,Z -42.871,A -90.000,B 90.000,C 0.000} C_DIS
LIN {X 117.651,Y -23.308,Z -43.202,A -90.000,B 90.000,C 0.000} C_DIS
LIN {X 117.607,Y -23.308,Z -43.727,A -90.000,B 90.000,C 0.000} C_DIS
LIN {X 117.567,Y -23.308,Z -44.117,A -90.000,B 90.000,C 0.000} C_DIS
LIN {X 117.489,Y -23.308,Z -44.635,A -90.000,B 90.000,C 0.000} C_DIS
LIN {X 117.399,Y -23.308,Z -45.114,A -90.000,B 90.000,C 0.000} C_DIS
LIN {X 117.260,Y -23.308,Z -45.739,A -90.000,B 90.000,C 0.000} C_DIS
LIN {X 117.102,Y -23.308,Z -46.271,A -90.000,B 90.000,C 0.000} C_DIS
LIN {X 116.900,Y -23.308,Z -46.938,A -90.000,B 90.000,C 0.000} C_DIS
LIN {X 116.543,Y -23.308,Z -47.863,A -90.000,B 90.000,C 0.000} C_DIS
LIN {X 116.372,Y -23.308,Z -48.278,A -90.000,B 90.000,C 0.000} C_DIS
LIN {X 115.873,Y -23.308,Z -49.350,A -90.000,B 90.000,C 0.000} C_DIS
LIN {X 115.226,Y -23.308,Z -50.643,A -90.000,B 90.000,C 0.000} C_DIS
LIN {X 114.622,Y -23.308,Z -51.838,A -90.000,B 90.000,C 0.000} C_DIS
LIN {X 113.941,Y -23.308,Z -53.229,A -90.000,B 90.000,C 0.000} C_DIS
LIN {X 113.276,Y -23.308,Z -54.687,A -90.000,B 90.000,C 0.000} C_DIS
LIN {X 112.865,Y -23.308,Z -55.672,A -90.000,B 90.000,C 0.000} C_DIS
LIN {X 112.799,Y -23.308,Z -55.830,A -90.000,B 90.000,C 0.000} C_DIS
LIN {X 112.213,Y -23.308,Z -57.388,A -90.000,B 90.000,C 0.000} C_DIS
LIN {X 111.674,Y -23.308,Z -59.009,A -90.000,B 90.000,C 0.000} C_DIS
LIN {X 111.260,Y -23.308,Z -60.445,A -90.000,B 90.000,C 0.000} C_DIS
LIN {X 110.695,Y -23.308,Z -62.513,A -90.000,B 90.000,C 0.000} C_DIS
LIN {X 110.151,Y -23.308,Z -64.443,A -90.000,B 90.000,C 0.000} C_DIS
LIN {X 110.021,Y -23.308,Z -64.879,A -90.000,B 90.000,C 0.000} C_DIS
LIN {X 109.345,Y -23.308,Z -67.050,A -90.000,B 90.000,C 0.000} C_DIS
LIN {X 108.519,Y -23.308,Z -69.358,A -90.000,B 90.000,C 0.000} C_DIS
LIN {X 107.578,Y -23.308,Z -71.726,A -90.000,B 90.000,C 0.000} C_DIS
LIN {X 107.403,Y -23.308,Z -72.150,A -90.000,B 90.000,C 0.000} C_DIS
LIN {X 106.414,Y -23.308,Z -74.420,A -90.000,B 90.000,C 0.000} C_DIS
LIN {X 105.411,Y -23.308,Z -76.516,A -90.000,B 90.000,C 0.000} C_DIS
LIN {X 104.209,Y -23.308,Z -78.763,A -90.000,B 90.000,C 0.000} C_DIS
LIN {X 103.931,Y -23.308,Z -79.244,A -90.000,B 90.000,C 0.000} C_DIS
LIN {X 103.058,Y -23.308,Z -80.726,A -90.000,B 90.000,C 0.000} C_DIS
LIN {X 102.198,Y -23.308,Z -82.078,A -90.000,B 90.000,C 0.000} C_DIS
LIN {X 99.737,Y -23.308,Z -85.762,A -90.000,B 90.000,C 0.000} C_DIS
LIN {X 99.871,Y -23.308,Z -87.489,A -90.000,B 90.000,C 0.000} C_DIS
LIN {X 100.012,Y -23.308,Z -89.494,A -90.000,B 90.000,C 0.000} C_DIS
LIN {X 100.049,Y -23.308,Z -90.038,A -90.000,B 90.000,C 0.000} C_DIS
LIN {X 100.093,Y -23.308,Z -90.499,A -90.000,B 90.000,C 0.000} C_DIS
LIN {X 100.108,Y -23.308,Z -90.704,A -90.000,B 90.000,C 0.000} C_DIS
LIN {X 100.173,Y -23.308,Z -91.769,A -90.000,B 90.000,C 0.000} C_DIS
LIN {X 100.205,Y -23.308,Z -92.178,A -90.000,B 90.000,C 0.000} C_DIS
LIN {X 100.236,Y -23.308,Z -92.421,A -90.000,B 90.000,C 0.000} C_DIS
LIN {X 100.261,Y -23.308,Z -92.907,A -90.000,B 90.000,C 0.000} C_DIS
LIN {X 100.247,Y -23.308,Z -93.625,A -90.000,B 90.000,C 0.000} C_DIS
LIN {X 100.276,Y -23.308,Z -94.544,A -90.000,B 90.000,C 0.000} C_DIS
LIN {X 100.265,Y -23.308,Z -94.867,A -90.000,B 90.000,C 0.000} C_DIS
LIN {X 100.225,Y -23.308,Z -95.634,A -90.000,B 90.000,C 0.000} C_DIS
LIN {X 100.234,Y -23.308,Z -95.942,A -90.000,B 90.000,C 0.000} C_DIS
LIN {X 100.223,Y -23.308,Z -96.265,A -90.000,B 90.000,C 0.000} C_DIS
LIN {X 100.177,Y -23.308,Z -96.904,A -90.000,B 90.000,C 0.000} C_DIS
LIN {X 100.184,Y -23.308,Z -98.220,A -90.000,B 90.000,C 0.000} C_DIS
LIN {X 100.184,Y -23.308,Z -98.382,A -90.000,B 90.000,C 0.000} C_DIS
LIN {X 100.165,Y -23.308,Z -98.791,A -90.000,B 90.000,C 0.000} C_DIS
LIN {X 100.149,Y -23.308,Z -99.048,A -90.000,B 90.000,C 0.000} C_DIS
LIN {X 100.161,Y -23.308,Z -99.891,A -90.000,B 90.000,C 0.000} C_DIS
LIN {X 100.143,Y -23.308,Z -100.300,A -90.000,B 90.000,C 0.000} C_DIS
LIN {X 100.118,Y -23.308,Z -100.671,A -90.000,B 90.000,C 0.000} C_DIS
LIN {X 100.138,Y -23.308,Z -101.379,A -90.000,B 90.000,C 0.000} C_DIS
LIN {X 100.117,Y -23.308,Z -101.951,A -90.000,B 90.000,C 0.000} C_DIS
LIN {X 100.106,Y -23.308,Z -102.199,A -90.000,B 90.000,C 0.000} C_DIS
LIN {X 100.151,Y -23.308,Z -103.037,A -90.000,B 90.000,C 0.000} C_DIS
LIN {X 100.149,Y -23.308,Z -103.540,A -90.000,B 90.000,C 0.000} C_DIS
LIN {X 100.171,Y -23.308,Z -103.833,A -90.000,B 90.000,C 0.000} C_DIS
LIN {X 100.239,Y -23.308,Z -104.465,A -90.000,B 90.000,C 0.000} C_DIS
LIN {X 100.318,Y -23.308,Z -105.016,A -90.000,B 90.000,C 0.000} C_DIS
LIN {X 100.367,Y -23.308,Z -105.327,A -90.000,B 90.000,C 0.000} C_DIS
LIN {X 100.532,Y -23.308,Z -106.263,A -90.000,B 90.000,C 0.000} C_DIS
LIN {X 100.802,Y -23.308,Z -107.935,A -90.000,B 90.000,C 0.000} C_DIS
LIN {X 100.844,Y -23.308,Z -108.306,A -90.000,B 90.000,C 0.000} C_DIS
LIN {X 100.972,Y -23.308,Z -109.350,A -90.000,B 90.000,C 0.000} C_DIS
LIN {X 101.005,Y -23.308,Z -109.725,A -90.000,B 90.000,C 0.000} C_DIS
LIN {X 101.132,Y -23.308,Z -110.977,A -90.000,B 90.000,C 0.000} C_DIS
LIN {X 101.167,Y -23.308,Z -111.428,A -90.000,B 90.000,C 0.000} C_DIS
LIN {X 101.297,Y -23.308,Z -112.823,A -90.000,B 90.000,C 0.000} C_DIS
LIN {X 101.309,Y -23.308,Z -112.981,A -90.000,B 90.000,C 0.000} C_DIS
LIN {X 101.502,Y -23.308,Z -115.034,A -90.000,B 90.000,C 0.000} C_DIS
LIN {X 101.691,Y -23.308,Z -116.950,A -90.000,B 90.000,C 0.000} C_DIS
LIN {X 101.702,Y -23.308,Z -117.081,A -90.000,B 90.000,C 0.000} C_DIS
LIN {X 101.895,Y -23.308,Z -119.127,A -90.000,B 90.000,C 0.000} C_DIS
LIN {X 101.919,Y -23.308,Z -119.442,A -90.000,B 90.000,C 0.000} C_DIS
LIN {X 102.074,Y -23.308,Z -121.348,A -90.000,B 90.000,C 0.000} C_DIS
LIN {X 102.219,Y -23.308,Z -123.710,A -90.000,B 90.000,C 0.000} C_DIS
LIN {X 102.272,Y -23.308,Z -124.746,A -90.000,B 90.000,C 0.000} C_DIS
LIN {X 102.343,Y -23.308,Z -127.095,A -90.000,B 90.000,C 0.000} C_DIS
LIN {X 102.340,Y -23.308,Z -127.283,A -90.000,B 90.000,C 0.000} C_DIS
LIN {X 102.342,Y -23.308,Z -129.537,A -90.000,B 90.000,C 0.000} C_DIS
LIN {X 102.338,Y -23.308,Z -129.695,A -90.000,B 90.000,C 0.000} C_DIS
LIN {X 102.325,Y -23.308,Z -130.053,A -90.000,B 90.000,C 0.000} C_DIS
LIN {X 102.274,Y -23.308,Z -132.267,A -90.000,B 90.000,C 0.000} C_DIS
LIN {X 102.247,Y -23.308,Z -132.794,A -90.000,B 90.000,C 0.000} C_DIS
LIN {X 102.154,Y -23.308,Z -135.105,A -90.000,B 90.000,C 0.000} C_DIS
LIN {X 102.014,Y -23.308,Z -137.840,A -90.000,B 90.000,C 0.000} C_DIS
LIN {X 101.781,Y -23.308,Z -141.760,A -90.000,B 90.000,C 0.000} C_DIS
LIN {X 101.496,Y -23.308,Z -145.941,A -90.000,B 90.000,C 0.000} C_DIS
LIN {X 101.254,Y -23.308,Z -149.133,A -90.000,B 90.000,C 0.000} C_DIS
LIN {X 101.037,Y -23.308,Z -151.660,A -90.000,B 90.000,C 0.000} C_DIS
LIN {X 100.950,Y -23.308,Z -152.845,A -90.000,B 90.000,C 0.000} C_DIS
LIN {X 100.914,Y -23.308,Z -153.267,A -90.000,B 90.000,C 0.000} C_DIS
LIN {X 100.731,Y -23.308,Z -155.213,A -90.000,B 90.000,C 0.000} C_DIS
LIN {X 100.628,Y -23.308,Z -156.544,A -90.000,B 90.000,C 0.000} C_DIS
LIN {X 100.592,Y -23.308,Z -156.966,A -90.000,B 90.000,C 0.000} C_DIS
LIN {X 100.423,Y -23.308,Z -158.631,A -90.000,B 90.000,C 0.000} C_DIS
LIN {X 100.278,Y -23.308,Z -160.414,A -90.000,B 90.000,C 0.000} C_DIS
LIN {X 100.257,Y -23.308,Z -160.663,A -90.000,B 90.000,C 0.000} C_DIS
LIN {X 100.197,Y -23.308,Z -161.204,A -90.000,B 90.000,C 0.000} C_DIS
LIN {X 99.946,Y -23.308,Z -164.195,A -90.000,B 90.000,C 0.000} C_DIS
LIN {X 99.596,Y -23.308,Z -167.947,A -90.000,B 90.000,C 0.000} C_DIS
LIN {X 99.230,Y -23.308,Z -171.649,A -90.000,B 90.000,C 0.000} C_DIS
LIN {X 99.135,Y -23.308,Z -172.558,A -90.000,B 90.000,C 0.000} C_DIS
LIN {X 98.888,Y -23.308,Z -174.853,A -90.000,B 90.000,C 0.000} C_DIS
LIN {X 98.857,Y -23.308,Z -175.182,A -90.000,B 90.000,C 0.000} C_DIS
LIN {X 98.605,Y -23.308,Z -177.435,A -90.000,B 90.000,C 0.000} C_DIS
LIN {X 98.546,Y -23.308,Z -178.060,A -90.000,B 90.000,C 0.000} C_DIS
LIN {X 98.387,Y -23.308,Z -179.441,A -90.000,B 90.000,C 0.000} C_DIS
LIN {X 98.235,Y -23.308,Z -180.930,A -90.000,B 90.000,C 0.000} C_DIS
LIN {X 98.126,Y -23.308,Z -181.853,A -90.000,B 90.000,C 0.000} C_DIS
LIN {X 97.942,Y -23.308,Z -183.566,A -90.000,B 90.000,C 0.000} C_DIS
LIN {X 97.875,Y -23.308,Z -184.137,A -90.000,B 90.000,C 0.000} C_DIS
LIN {X 97.394,Y -23.308,Z -188.511,A -90.000,B 90.000,C 0.000} C_DIS
LIN {X 97.125,Y -23.308,Z -190.962,A -90.000,B 90.000,C 0.000} C_DIS
LIN {X 96.829,Y -23.308,Z -193.288,A -90.000,B 90.000,C 0.000} C_DIS
LIN {X 96.779,Y -23.308,Z -193.645,A -90.000,B 90.000,C 0.000} C_DIS
LIN {X 96.266,Y -23.308,Z -196.628,A -90.000,B 90.000,C 0.000} C_DIS
LIN {X 95.529,Y -23.308,Z -200.180,A -90.000,B 90.000,C 0.000} C_DIS
LIN {X 95.435,Y -23.308,Z -200.606,A -90.000,B 90.000,C 0.000} C_DIS
LIN {X 94.275,Y -23.308,Z -205.314,A -90.000,B 90.000,C 0.000} C_DIS
LIN {X 93.124,Y -23.308,Z -209.715,A -90.000,B 90.000,C 0.000} C_DIS
LIN {X 92.883,Y -23.308,Z -210.670,A -90.000,B 90.000,C 0.000} C_DIS
LIN {X 91.737,Y -23.308,Z -214.952,A -90.000,B 90.000,C 0.000} C_DIS
LIN {X 91.354,Y -23.308,Z -216.446,A -90.000,B 90.000,C 0.000} C_DIS
LIN {X 90.298,Y -23.308,Z -220.397,A -90.000,B 90.000,C 0.000} C_DIS
LIN {X 89.457,Y -23.308,Z -223.605,A -90.000,B 90.000,C 0.000} C_DIS
LIN {X 88.878,Y -23.308,Z -225.862,A -90.000,B 90.000,C 0.000} C_DIS
LIN {X 88.267,Y -23.308,Z -228.099,A -90.000,B 90.000,C 0.000} C_DIS
LIN {X 87.377,Y -23.308,Z -231.386,A -90.000,B 90.000,C 0.000} C_DIS
LIN {X 86.871,Y -23.308,Z -233.073,A -90.000,B 90.000,C 0.000} C_DIS
LIN {X 85.665,Y -23.308,Z -237.135,A -90.000,B 90.000,C 0.000} C_DIS
LIN {X 85.527,Y -23.308,Z -237.550,A -90.000,B 90.000,C 0.000} C_DIS
LIN {X 85.112,Y -23.308,Z -238.770,A -90.000,B 90.000,C 0.000} C_DIS
LIN {X 83.516,Y -23.308,Z -243.561,A -90.000,B 90.000,C 0.000} C_DIS
LIN {X 83.516,Y -60.000,Z -243.561,A -90.000,B 90.000,C 0.000} C_DIS
LIN {X 100.054,Y -60.000,Z -90.033,A -90.000,B 90.000,C 0.000} C_DIS
LIN {X 100.054,Y -21.308,Z -90.033,A -90.000,B 90.000,C 0.000} C_DIS
LIN {X 100.213,Y -21.311,Z -90.847,A -90.000,B 90.000,C 0.000} C_DIS
LIN {X 100.321,Y -21.315,Z -91.543,A -90.000,B 90.000,C 0.000} C_DIS
LIN {X 100.421,Y -21.317,Z -92.378,A -90.000,B 90.000,C 0.000} C_DIS
LIN {X 100.447,Y -21.319,Z -92.522,A -90.000,B 90.000,C 0.000} C_DIS
LIN {X 100.520,Y -21.326,Z -93.005,A -90.000,B 90.000,C 0.000} C_DIS
LIN {X 100.544,Y -21.330,Z -93.486,A -90.000,B 90.000,C 0.000} C_DIS
LIN {X 100.551,Y -21.331,Z -93.765,A -90.000,B 90.000,C 0.000} C_DIS
LIN {X 100.613,Y -21.337,Z -94.493,A -90.000,B 90.000,C 0.000} C_DIS
LIN {X 100.635,Y -21.344,Z -94.940,A -90.000,B 90.000,C 0.000} C_DIS
LIN {X 100.632,Y -21.344,Z -95.039,A -90.000,B 90.000,C 0.000} C_DIS
LIN {X 100.644,Y -21.353,Z -95.624,A -90.000,B 90.000,C 0.000} C_DIS
LIN {X 100.651,Y -21.352,Z -95.956,A -90.000,B 90.000,C 0.000} C_DIS
LIN {X 100.663,Y -21.357,Z -96.218,A -90.000,B 90.000,C 0.000} C_DIS
LIN {X 100.659,Y -21.367,Z -96.918,A -90.000,B 90.000,C 0.000} C_DIS
LIN {X 100.659,Y -21.367,Z -97.173,A -90.000,B 90.000,C 0.000} C_DIS
LIN {X 100.670,Y -21.369,Z -97.321,A -90.000,B 90.000,C 0.000} C_DIS
LIN {X 100.707,Y -21.378,Z -98.092,A -90.000,B 90.000,C 0.000} C_DIS
LIN {X 100.709,Y -21.379,Z -98.399,A -90.000,B 90.000,C 0.000} C_DIS
LIN {X 100.711,Y -21.384,Z -98.816,A -90.000,B 90.000,C 0.000} C_DIS
LIN {X 100.729,Y -21.394,Z -99.063,A -90.000,B 90.000,C 0.000} C_DIS
LIN {X 100.750,Y -21.399,Z -99.498,A -90.000,B 90.000,C 0.000} C_DIS
LIN {X 100.755,Y -21.399,Z -99.918,A -90.000,B 90.000,C 0.000} C_DIS
LIN {X 100.757,Y -21.405,Z -100.328,A -90.000,B 90.000,C 0.000} C_DIS
LIN {X 100.770,Y -21.413,Z -100.479,A -90.000,B 90.000,C 0.000} C_DIS
LIN {X 100.780,Y -21.421,Z -100.720,A -90.000,B 90.000,C 0.000} C_DIS
LIN {X 100.791,Y -21.422,Z -100.949,A -90.000,B 90.000,C 0.000} C_DIS
LIN {X 100.803,Y -21.423,Z -101.445,A -90.000,B 90.000,C 0.000} C_DIS
LIN {X 100.809,Y -21.431,Z -101.836,A -90.000,B 90.000,C 0.000} C_DIS
LIN {X 100.842,Y -21.448,Z -102.206,A -90.000,B 90.000,C 0.000} C_DIS
LIN {X 100.887,Y -21.449,Z -103.070,A -90.000,B 90.000,C 0.000} C_DIS
LIN {X 100.893,Y -21.451,Z -103.215,A -90.000,B 90.000,C 0.000} C_DIS
LIN {X 100.919,Y -21.463,Z -103.512,A -90.000,B 90.000,C 0.000} C_DIS
LIN {X 100.960,Y -21.465,Z -103.903,A -90.000,B 90.000,C 0.000} C_DIS
LIN {X 100.977,Y -21.465,Z -104.066,A -90.000,B 90.000,C 0.000} C_DIS
LIN {X 101.020,Y -21.469,Z -104.386,A -90.000,B 90.000,C 0.000} C_DIS
LIN {X 101.135,Y -21.469,Z -105.153,A -90.000,B 90.000,C 0.000} C_DIS
LIN {X 101.348,Y -21.468,Z -106.401,A -90.000,B 90.000,C 0.000} C_DIS
LIN {X 101.447,Y -21.468,Z -107.019,A -90.000,B 90.000,C 0.000} C_DIS
LIN {X 101.577,Y -21.466,Z -107.852,A -90.000,B 90.000,C 0.000} C_DIS
LIN {X 101.601,Y -21.469,Z -108.021,A -90.000,B 90.000,C 0.000} C_DIS
LIN {X 101.757,Y -21.471,Z -109.254,A -90.000,B 90.000,C 0.000} C_DIS
LIN {X 101.805,Y -21.476,Z -109.692,A -90.000,B 90.000,C 0.000} C_DIS
LIN {X 101.910,Y -21.480,Z -110.612,A -90.000,B 90.000,C 0.000} C_DIS
LIN {X 101.945,Y -21.482,Z -110.914,A -90.000,B 90.000,C 0.000} C_DIS
LIN {X 102.001,Y -21.488,Z -111.452,A -90.000,B 90.000,C 0.000} C_DIS
LIN {X 102.100,Y -21.494,Z -112.370,A -90.000,B 90.000,C 0.000} C_DIS
LIN {X 102.144,Y -21.497,Z -112.759,A -90.000,B 90.000,C 0.000} C_DIS
LIN {X 102.334,Y -21.511,Z -114.520,A -90.000,B 90.000,C 0.000} C_DIS
LIN {X 102.373,Y -21.515,Z -114.854,A -90.000,B 90.000,C 0.000} C_DIS
LIN {X 102.613,Y -21.530,Z -117.002,A -90.000,B 90.000,C 0.000} C_DIS
LIN {X 102.834,Y -21.544,Z -119.057,A -90.000,B 90.000,C 0.000} C_DIS
LIN {X 102.877,Y -21.549,Z -119.480,A -90.000,B 90.000,C 0.000} C_DIS
LIN {X 103.051,Y -21.564,Z -121.288,A -90.000,B 90.000,C 0.000} C_DIS
LIN {X 103.094,Y -21.572,Z -121.762,A -90.000,B 90.000,C 0.000} C_DIS
LIN {X 103.127,Y -21.577,Z -122.172,A -90.000,B 90.000,C 0.000} C_DIS
LIN {X 103.229,Y -21.588,Z -123.522,A -90.000,B 90.000,C 0.000} C_DIS
LIN {X 103.280,Y -21.596,Z -124.210,A -90.000,B 90.000,C 0.000} C_DIS
LIN {X 103.306,Y -21.597,Z -124.696,A -90.000,B 90.000,C 0.000} C_DIS
LIN {X 103.417,Y -21.621,Z -127.063,A -90.000,B 90.000,C 0.000} C_DIS
LIN {X 103.451,Y -21.644,Z -129.481,A -90.000,B 90.000,C 0.000} C_DIS
LIN {X 103.451,Y -21.644,Z -129.538,A -90.000,B 90.000,C 0.000} C_DIS
LIN {X 103.443,Y -21.650,Z -130.086,A -90.000,B 90.000,C 0.000} C_DIS
LIN {X 103.420,Y -21.667,Z -132.141,A -90.000,B 90.000,C 0.000} C_DIS
LIN {X 103.415,Y -21.667,Z -132.326,A -90.000,B 90.000,C 0.000} C_DIS
LIN {X 103.397,Y -21.673,Z -132.847,A -90.000,B 90.000,C 0.000} C_DIS
LIN {X 103.324,Y -21.687,Z -135.165,A -90.000,B 90.000,C 0.000} C_DIS
